C08987=1026.109,2.231,-95.350,167.487,46.558,158.592
C08988=1026.114,2.480,-95.365,167.491,46.555,158.592
C08989=1026.122,2.729,-95.379,167.493,46.552,158.592
C08990=1026.127,2.979,-95.393,167.495,46.549,158.592
C08991=1026.133,3.228,-95.408,167.498,46.546,158.592
C08992=1026.139,3.477,-95.423,167.501,46.544,158.592
C08993=1026.146,3.727,-95.438,167.503,46.541,158.591
C08994=1026.151,3.977,-95.452,167.506,46.538,158.591
C08995=1026.157,4.226,-95.467,167.509,46.535,158.591
C08996=1026.164,4.476,-95.481,167.511,46.533,158.591
C08997=1026.170,4.725,-95.496,167.514,46.530,158.590
C08998=1026.176,4.975,-95.510,167.516,46.527,158.590
C08999=1026.181,5.224,-95.525,167.519,46.524,158.590
C09000=1026.188,5.474,-95.540,167.522,46.521,158.590
C09001=1026.194,5.723,-95.555,167.524,46.519,158.590
C09002=1026.200,5.973,-95.568,167.527,46.516,158.589
C09003=1026.207,6.222,-95.583,167.530,46.513,158.589
C09004=1026.213,6.471,-95.598,167.532,46.510,158.589
C09005=1026.219,6.721,-95.612,167.534,46.507,158.589
C09006=1026.225,6.971,-95.627,167.538,46.504,158.589
C09007=1026.231,7.219,-95.642,167.540,46.502,158.588
C09008=1026.237,7.470,-95.656,167.542,46.499,158.588
C09009=1026.244,7.719,-95.671,167.545,46.496,158.588
C09010=1026.249,7.968,-95.686,167.548,46.493,158.588
C09011=1026.256,8.218,-95.701,167.550,46.490,158.587
C09012=1026.262,8.468,-95.716,167.553,46.487,158.587
C09013=1026.268,8.717,-95.730,167.555,46.485,158.587
C09014=1026.274,8.967,-95.744,167.559,46.482,158.587
C09015=1026.280,9.217,-95.759,167.561,46.479,158.587
C09016=1026.286,9.466,-95.774,167.563,46.477,158.586
C09017=1026.293,9.715,-95.789,167.567,46.474,158.586
C09018=1026.299,9.965,-95.804,167.569,46.471,158.586
C09019=1026.306,10.214,-95.818,167.571,46.468,158.586
C09020=1026.312,10.463,-95.833,167.574,46.465,158.586
C09021=1026.318,10.713,-95.848,167.577,46.462,158.585
C09022=1026.325,10.962,-95.863,167.579,46.459,158.585
C09023=1026.331,11.246,-95.880,167.582,46.456,158.585
C09024=1026.339,11.530,-95.896,167.585,46.453,158.585
C09025=1026.346,11.815,-95.914,167.588,46.450,158.584
C09026=1026.353,12.098,-95.930,167.591,46.446,158.584
C09027=1026.359,12.348,-95.945,167.594,46.443,158.584
C09028=1026.365,12.598,-95.960,167.596,46.440,158.584
C09029=1026.371,12.847,-95.974,167.599,46.437,158.583
C09030=1026.377,13.097,-95.989,167.601,46.435,158.583
C09031=1026.384,13.347,-96.004,167.604,46.432,158.583
C09032=1026.390,13.596,-96.019,167.607,46.429,158.583
C09033=1026.396,13.845,-96.034,167.609,46.426,158.583
C09034=1026.402,14.094,-96.049,167.611,46.423,158.582
C09035=1026.408,14.344,-96.064,167.614,46.421,158.582
C09036=1026.415,14.594,-96.079,167.617,46.418,158.582
C09037=1026.420,14.843,-96.094,167.619,46.415,158.582
C09038=1026.427,15.093,-96.109,167.622,46.413,158.581
C09039=1026.432,15.343,-96.124,167.625,46.410,158.581
C09040=1026.439,15.592,-96.139,167.627,46.407,158.581
C09041=1026.445,15.841,-96.155,167.629,46.404,158.581
C09042=1026.451,16.090,-96.170,167.632,46.401,158.581
C09043=1026.458,16.340,-96.185,167.635,46.399,158.581
C09044=1026.463,16.590,-96.200,167.637,46.396,158.580
C09045=1026.470,16.839,-96.215,167.640,46.394,158.580
C09046=1026.475,17.088,-96.230,167.643,46.391,158.580
C09047=1026.482,17.337,-96.245,167.645,46.388,158.580
C09048=1026.488,17.587,-96.261,167.647,46.385,158.579
C09049=1026.494,17.837,-96.276,167.650,46.382,158.579
C09050=1026.500,18.087,-96.291,167.653,46.379,158.579
C09051=1026.507,18.335,-96.306,167.655,46.376,158.579
C09052=1026.512,18.585,-96.322,167.657,46.374,158.578
C09053=1026.519,18.835,-96.337,167.661,46.371,158.578
C09054=1026.525,19.084,-96.351,167.663,46.369,158.578
C09055=1026.532,19.333,-96.367,167.665,46.366,158.578
C09056=1026.537,19.583,-96.383,167.668,46.363,158.578
C09057=1026.543,19.832,-96.397,167.671,46.360,158.577
C09058=1026.549,20.082,-96.412,167.673,46.357,158.577
C09059=1026.555,20.331,-96.428,167.675,46.354,158.577
C09060=1026.562,20.581,-96.443,167.678,46.352,158.577
C09061=1026.567,20.831,-96.459,167.681,46.349,158.577
C09062=1026.574,21.080,-96.475,167.683,46.347,158.576
C09063=1026.581,21.330,-96.490,167.686,46.344,158.576
C09064=1026.586,21.578,-96.505,167.688,46.341,158.576
C09065=1026.592,21.828,-96.520,167.691,46.338,158.576
C09066=1026.598,22.078,-96.536,167.693,46.335,158.575
C09067=1026.605,22.327,-96.552,167.696,46.333,158.575
C09068=1026.611,22.577,-96.567,167.698,46.330,158.575
C09069=1026.617,22.827,-96.582,167.701,46.327,158.575
C09070=1026.623,23.076,-96.598,167.704,46.325,158.575
C09071=1026.629,23.326,-96.613,167.706,46.322,158.574
C09072=1026.635,23.574,-96.629,167.708,46.319,158.574
C09073=1026.641,23.824,-96.644,167.711,46.316,158.574
C09074=1026.647,24.073,-96.660,167.714,46.313,158.574
C09075=1026.654,24.323,-96.675,167.716,46.311,158.573
C09076=1026.659,24.573,-96.690,167.718,46.308,158.573
C09077=1026.666,24.822,-96.706,167.721,46.305,158.573
C09078=1026.672,25.071,-96.721,167.724,46.302,158.573
C09079=1026.678,25.321,-96.737,167.726,46.299,158.573
C09080=1026.685,25.570,-96.752,167.729,46.296,158.572
C09081=1026.691,25.820,-96.768,167.732,46.294,158.572
C09082=1026.697,26.069,-96.783,167.734,46.292,158.572
C09083=1026.703,26.319,-96.800,167.736,46.289,158.572
C09084=1026.709,26.568,-96.814,167.739,46.286,158.572
C09085=1026.716,26.817,-96.830,167.742,46.283,158.571
C09086=1026.721,27.067,-96.845,167.744,46.280,158.571
C09087=1026.729,27.352,-96.863,167.747,46.277,158.571
C09088=1026.736,27.637,-96.881,167.749,46.274,158.570
C09089=1026.742,27.923,-96.900,167.752,46.271,158.570
C09090=1026.750,28.208,-96.917,167.756,46.268,158.570
C09091=1026.756,28.458,-96.933,167.758,46.265,158.570
C09092=1026.761,28.707,-96.949,167.760,46.262,158.570
C09093=1026.768,28.956,-96.965,167.762,46.260,158.569
C09094=1026.774,29.206,-96.980,167.766,46.257,158.569
C09095=1026.780,29.455,-96.996,167.768,46.254,158.569
C09096=1026.786,29.705,-97.012,167.770,46.252,158.569
C09097=1026.792,29.955,-97.028,167.773,46.249,158.569
C09098=1026.799,30.204,-97.043,167.776,46.246,158.568
C09099=1026.805,30.453,-97.060,167.778,46.243,158.568
C09100=1026.810,30.703,-97.075,167.780,46.240,158.568
C09101=1026.817,30.952,-97.091,167.783,46.238,158.568
C09102=1026.823,31.201,-97.107,167.785,46.236,158.567
C09103=1026.829,31.451,-97.123,167.788,46.233,158.567
C09104=1026.835,31.700,-97.138,167.791,46.230,158.567
C09105=1026.841,31.950,-97.155,167.793,46.227,158.567
C09106=1026.847,32.199,-97.171,167.795,46.224,158.567
C09107=1026.854,32.449,-97.186,167.798,46.221,158.566
C09108=1026.860,32.698,-97.202,167.801,46.219,158.566
C09109=1026.866,32.948,-97.218,167.803,46.216,158.566
C09110=1026.872,33.197,-97.234,167.805,46.213,158.566
C09111=1026.878,33.447,-97.249,167.808,46.211,158.565
C09112=1026.884,33.696,-97.266,167.811,46.208,158.565
C09113=1026.891,33.945,-97.281,167.813,46.205,158.565
C09114=1026.896,34.194,-97.298,167.815,46.203,158.565
C09115=1026.904,34.444,-97.314,167.818,46.200,158.565
C09116=1026.909,34.694,-97.329,167.821,46.197,158.564
C09117=1026.915,34.943,-97.345,167.823,46.194,158.564
C09118=1026.922,35.192,-97.361,167.825,46.191,158.564
C09119=1026.928,35.442,-97.377,167.828,46.189,158.564
C09120=1026.934,35.691,-97.394,167.830,46.186,158.563
C09121=1026.941,35.940,-97.409,167.833,46.183,158.563
C09122=1026.946,36.190,-97.425,167.836,46.180,158.563
C09123=1026.952,36.439,-97.441,167.838,46.177,158.563
C09124=1026.958,36.689,-97.457,167.840,46.175,158.562
C09125=1026.965,36.938,-97.473,167.843,46.172,158.562
C09126=1026.971,37.188,-97.490,167.846,46.170,158.562
C09127=1026.977,37.437,-97.506,167.848,46.167,158.562
C09128=1026.983,37.687,-97.522,167.850,46.164,158.562
C09129=1026.989,37.936,-97.538,167.853,46.161,158.561
C09130=1026.995,38.185,-97.555,167.856,46.158,158.561
C09131=1027.001,38.435,-97.571,167.858,46.156,158.561
C09132=1027.008,38.684,-97.587,167.861,46.153,158.561
C09133=1027.014,38.933,-97.603,167.863,46.151,158.560
C09134=1027.020,39.182,-97.619,167.865,46.148,158.560
C09135=1027.026,39.432,-97.635,167.867,46.145,158.560
C09136=1027.032,39.682,-97.652,167.871,46.142,158.560
C09137=1027.038,39.931,-97.668,167.873,46.140,158.560
C09138=1027.044,40.180,-97.684,167.875,46.137,158.559
C09139=1027.050,40.430,-97.701,167.878,46.135,158.559
C09140=1027.056,40.679,-97.717,167.880,46.132,158.559
C09141=1027.062,40.928,-97.733,167.883,46.129,158.559
C09142=1027.068,41.178,-97.749,167.885,46.126,158.558
C09143=1027.075,41.428,-97.766,167.888,46.123,158.558
C09144=1027.081,41.677,-97.782,167.890,46.121,158.558
C09145=1027.087,41.926,-97.798,167.892,46.119,158.558
C09146=1027.093,42.176,-97.814,167.895,46.116,158.558
C09147=1027.099,42.425,-97.831,167.898,46.113,158.557
C09148=1027.105,42.674,-97.847,167.900,46.110,158.557
C09149=1027.112,42.924,-97.864,167.902,46.107,158.557
C09150=1027.118,43.173,-97.880,167.905,46.105,158.557
C09151=1027.124,43.459,-97.899,167.908,46.102,158.556
C09152=1027.131,43.744,-97.918,167.910,46.099,158.556
C09153=1027.138,44.029,-97.937,167.914,46.096,158.556
C09154=1027.145,44.315,-97.956,167.916,46.093,158.556
C09155=1027.151,44.565,-97.973,167.919,46.090,158.556
C09156=1027.157,44.813,-97.990,167.921,46.088,158.555
C09157=1027.163,45.063,-98.006,167.924,46.085,158.555
C09158=1027.169,45.312,-98.022,167.926,46.083,158.555
C09159=1027.175,45.562,-98.039,167.928,46.080,158.555
C09160=1027.181,45.811,-98.056,167.931,46.077,158.554
C09161=1027.187,46.060,-98.073,167.933,46.075,158.554
C09162=1027.193,46.310,-98.089,167.936,46.072,158.554
C09163=1027.199,46.559,-98.105,167.939,46.070,158.554
C09164=1027.205,46.809,-98.123,167.941,46.067,158.554
C09165=1027.211,47.058,-98.139,167.943,46.064,158.553
C09166=1027.217,47.308,-98.156,167.946,46.062,158.553
C09167=1027.223,47.556,-98.173,167.948,46.059,158.553
C09168=1027.230,47.806,-98.189,167.950,46.057,158.553
C09169=1027.235,48.056,-98.206,167.953,46.054,158.552
C09170=1027.241,48.305,-98.223,167.956,46.051,158.552
C09171=1027.247,48.554,-98.239,167.958,46.048,158.552
C09172=1027.253,48.803,-98.256,167.961,46.046,158.552
C09173=1027.260,49.053,-98.273,167.963,46.043,158.552
C09174=1027.265,49.303,-98.290,167.965,46.041,158.551
C09175=1027.271,49.552,-98.306,167.967,46.038,158.551
C09176=1027.277,49.801,-98.323,167.971,46.035,158.551
C09177=1027.284,50.051,-98.340,167.973,46.033,158.551
C09178=1027.290,50.299,-98.357,167.975,46.030,158.550
C09179=1027.295,50.549,-98.373,167.978,46.027,158.550
C09180=1027.302,50.799,-98.390,167.980,46.025,158.550
C09181=1027.308,51.048,-98.407,167.982,46.022,158.550
C09182=1027.314,51.297,-98.423,167.984,46.019,158.549
C09183=1027.320,51.546,-98.440,167.988,46.016,158.549
C09184=1027.326,51.796,-98.457,167.990,46.014,158.549
C09185=1027.332,52.045,-98.474,167.992,46.011,158.549
C09186=1027.338,52.294,-98.491,167.995,46.009,158.549
C09187=1027.345,52.544,-98.507,167.997,46.006,158.548
C09188=1027.350,52.793,-98.525,167.999,46.003,158.548
C09189=1027.356,53.043,-98.541,168.002,46.000,158.548
C09190=1027.363,53.292,-98.558,168.005,45.997,158.548
C09191=1027.369,53.542,-98.575,168.007,45.995,158.547
C09192=1027.375,53.790,-98.592,168.009,45.993,158.547
C09193=1027.381,54.041,-98.609,168.012,45.990,158.547
C09194=1027.387,54.289,-98.626,168.014,45.987,158.547
C09195=1027.393,54.539,-98.642,168.017,45.984,158.547
C09196=1027.400,54.788,-98.659,168.020,45.982,158.546
C09197=1027.406,55.038,-98.676,168.022,45.979,158.546
C09198=1027.412,55.287,-98.693,168.024,45.976,158.546
C09199=1027.418,55.537,-98.710,168.026,45.973,158.545
C09200=1027.425,55.785,-98.727,168.030,45.970,158.545
C09201=1027.431,56.035,-98.745,168.032,45.968,158.545
C09202=1027.437,56.284,-98.761,168.034,45.965,158.545
C09203=1027.443,56.533,-98.778,168.036,45.962,158.544
C09204=1027.449,56.783,-98.795,168.039,45.960,158.544
C09205=1027.456,57.032,-98.812,168.041,45.957,158.544
C09206=1027.462,57.282,-98.829,168.044,45.954,158.544
C09207=1027.468,57.531,-98.846,168.047,45.952,158.544
C09208=1027.474,57.780,-98.863,168.049,45.949,158.543
C09209=1027.481,58.030,-98.879,168.051,45.946,158.543
C09210=1027.486,58.279,-98.897,168.053,45.944,158.543
C09211=1027.493,58.529,-98.914,168.057,45.941,158.543
C09212=1027.499,58.778,-98.931,168.059,45.938,158.542
C09213=1027.505,59.026,-98.948,168.061,45.935,158.542
C09214=1027.511,59.277,-98.965,168.064,45.932,158.542
C09215=1027.518,59.562,-98.984,168.067,45.929,158.542
C09216=1027.526,59.847,-99.004,168.069,45.926,158.541
C09217=1027.532,60.132,-99.023,168.072,45.923,158.541
C09218=1027.540,60.417,-99.042,168.075,45.919,158.541
C09219=1027.546,60.666,-99.060,168.077,45.917,158.540
C09220=1027.552,60.916,-99.077,168.080,45.914,158.540
C09221=1027.559,61.165,-99.094,168.082,45.911,158.540
C09222=1027.565,61.414,-99.111,168.085,45.908,158.540
C09223=1027.571,61.664,-99.128,168.087,45.906,158.539
C09224=1027.577,61.913,-99.145,168.090,45.903,158.539
C09225=1027.584,62.163,-99.162,168.092,45.900,158.539
C09226=1027.590,62.411,-99.179,168.094,45.897,158.539
C09227=1027.597,62.661,-99.196,168.097,45.894,158.538
C09228=1027.602,62.910,-99.214,168.100,45.892,158.538
C09229=1027.609,63.160,-99.231,168.102,45.889,158.538
C09230=1027.615,63.409,-99.247,168.104,45.886,158.538
C09231=1027.621,63.659,-99.265,168.107,45.884,158.537
C09232=1027.627,63.908,-99.282,168.110,45.881,158.537
C09233=1027.633,64.157,-99.300,168.112,45.879,158.537
C09234=1027.640,64.406,-99.317,168.115,45.876,158.537
C09235=1027.646,64.656,-99.335,168.117,45.873,158.537
C09236=1027.652,64.905,-99.352,168.119,45.870,158.536
C09237=1027.658,65.154,-99.370,168.121,45.868,158.536
C09238=1027.663,65.404,-99.387,168.125,45.865,158.536
C09239=1027.670,65.653,-99.404,168.127,45.862,158.536
C09240=1027.676,65.902,-99.422,168.129,45.859,158.535
C09241=1027.683,66.152,-99.439,168.132,45.857,158.535
C09242=1027.688,66.401,-99.457,168.134,45.855,158.535
C09243=1027.695,66.650,-99.474,168.136,45.852,158.535
C09244=1027.700,66.899,-99.491,168.139,45.849,158.534
C09245=1027.707,67.149,-99.509,168.142,45.846,158.534
C09246=1027.713,67.398,-99.526,168.144,45.843,158.534
C09247=1027.719,67.648,-99.544,168.146,45.841,158.534
C09248=1027.725,67.896,-99.561,168.149,45.838,158.533
C09249=1027.731,68.146,-99.579,168.151,45.835,158.533
C09250=1027.737,68.396,-99.597,168.153,45.833,158.533
C09251=1027.744,68.644,-99.614,168.157,45.830,158.533
C09252=1027.750,68.894,-99.632,168.159,45.828,158.533
C09253=1027.755,69.143,-99.650,168.161,45.825,158.532
C09254=1027.762,69.393,-99.667,168.163,45.822,158.532
C09255=1027.768,69.642,-99.684,168.166,45.819,158.532
C09256=1027.774,69.891,-99.702,168.168,45.817,158.532
C09257=1027.779,70.141,-99.720,168.171,45.815,158.531
C09258=1027.786,70.390,-99.737,168.173,45.812,158.531
C09259=1027.792,70.640,-99.755,168.176,45.809,158.531
C09260=1027.798,70.889,-99.773,168.178,45.806,158.531
C09261=1027.804,71.138,-99.791,168.181,45.804,158.530
C09262=1027.811,71.387,-99.808,168.183,45.801,158.530
C09263=1027.817,71.636,-99.826,168.185,45.799,158.530
C09264=1027.822,71.885,-99.844,168.188,45.796,158.530
C09265=1027.828,72.135,-99.862,168.190,45.793,158.529
C09266=1027.835,72.385,-99.879,168.193,45.791,158.529
C09267=1027.841,72.634,-99.897,168.195,45.788,158.529
C09268=1027.847,72.883,-99.915,168.198,45.785,158.529
C09269=1027.853,73.132,-99.933,168.200,45.783,158.529
C09270=1027.859,73.381,-99.951,168.203,45.780,158.528
C09271=1027.866,73.631,-99.968,168.205,45.778,158.528
C09272=1027.871,73.880,-99.986,168.207,45.775,158.528
C09273=1027.877,74.130,-100.004,168.210,45.772,158.528
C09274=1027.883,74.378,-100.022,168.213,45.769,158.527
C09275=1027.889,74.628,-100.040,168.215,45.767,158.527
C09276=1027.896,74.877,-100.057,168.217,45.764,158.527
C09277=1027.902,75.126,-100.075,168.220,45.762,158.527
C09278=1027.908,75.376,-100.093,168.222,45.759,158.526
C09279=1027.915,75.661,-100.113,168.225,45.756,158.526
C09280=1027.922,75.946,-100.134,168.228,45.753,158.526
C09281=1027.929,76.231,-100.154,168.231,45.750,158.526
C09282=1027.936,76.516,-100.175,168.234,45.746,158.525
C09283=1027.942,76.766,-100.193,168.236,45.744,158.525
C09284=1027.948,77.015,-100.211,168.238,45.742,158.525
C09285=1027.954,77.264,-100.229,168.241,45.739,158.525
C09286=1027.960,77.513,-100.246,168.243,45.736,158.524
C09287=1027.967,77.762,-100.265,168.246,45.733,158.524
C09288=1027.972,78.011,-100.282,168.248,45.730,158.524
C09289=1027.979,78.261,-100.300,168.251,45.728,158.524
C09290=1027.984,78.511,-100.320,168.253,45.726,158.523
C09291=1027.990,78.760,-100.337,168.256,45.723,158.523
C09292=1027.996,79.009,-100.356,168.258,45.720,158.523
C09293=1028.002,79.258,-100.374,168.260,45.718,158.523
C09294=1028.008,79.507,-100.392,168.263,45.716,158.522
C09295=1028.014,79.757,-100.410,168.265,45.713,158.522
C09296=1028.020,80.006,-100.428,168.268,45.710,158.522
C09297=1028.026,80.255,-100.446,168.270,45.707,158.522
C09298=1028.032,80.505,-100.464,168.273,45.705,158.522
C09299=1028.039,80.754,-100.483,168.275,45.703,158.521
C09300=1028.044,81.003,-100.500,168.278,45.700,158.521
C09301=1028.051,81.252,-100.519,168.280,45.697,158.521
C09302=1028.057,81.502,-100.537,168.282,45.694,158.520
C09303=1028.063,81.751,-100.556,168.285,45.692,158.520
C09304=1028.068,82.000,-100.574,168.288,45.689,158.520
C09305=1028.074,82.249,-100.592,168.290,45.687,158.520
C09306=1028.081,82.499,-100.610,168.292,45.684,158.520
C09307=1028.086,82.747,-100.629,168.295,45.681,158.519
C09308=1028.092,82.997,-100.647,168.297,45.679,158.519
C09309=1028.099,83.246,-100.665,168.299,45.677,158.519
C09310=1028.105,83.496,-100.683,168.302,45.674,158.519
C09311=1028.111,83.744,-100.701,168.305,45.671,158.518
C09312=1028.117,83.994,-100.719,168.307,45.668,158.518
C09313=1028.123,84.243,-100.738,168.310,45.666,158.518
C09314=1028.130,84.492,-100.757,168.312,45.663,158.518
C09315=1028.135,84.741,-100.774,168.314,45.661,158.518
C09316=1028.141,84.991,-100.793,168.317,45.658,158.517
C09317=1028.147,85.241,-100.811,168.320,45.655,158.517
C09318=1028.154,85.490,-100.830,168.322,45.653,158.517
C09319=1028.160,85.739,-100.848,168.325,45.650,158.517
C09320=1028.166,85.988,-100.866,168.327,45.647,158.516
C09321=1028.172,86.237,-100.885,168.329,45.645,158.516
C09322=1028.178,86.487,-100.903,168.332,45.642,158.516
C09323=1028.184,86.736,-100.921,168.335,45.640,158.516
C09324=1028.191,86.985,-100.940,168.337,45.637,158.515
C09325=1028.196,87.234,-100.958,168.339,45.634,158.515
C09326=1028.203,87.483,-100.976,168.342,45.631,158.515
C09327=1028.209,87.732,-100.996,168.344,45.629,158.515
C09328=1028.215,87.982,-101.014,168.346,45.626,158.514
C09329=1028.221,88.231,-101.032,168.350,45.623,158.514
C09330=1028.227,88.481,-101.050,168.352,45.620,158.514
C09331=1028.233,88.730,-101.068,168.354,45.618,158.514
C09332=1028.239,88.979,-101.087,168.357,45.616,158.513
C09333=1028.246,89.228,-101.106,168.359,45.613,158.513
C09334=1028.252,89.477,-101.124,168.361,45.610,158.513
C09335=1028.258,89.727,-101.143,168.364,45.607,158.513
C09336=1028.264,89.976,-101.162,168.367,45.605,158.512
C09337=1028.271,90.225,-101.180,168.369,45.603,158.512
C09338=1028.275,90.475,-101.198,168.372,45.600,158.512
C09339=1028.282,90.724,-101.217,168.374,45.597,158.512
C09340=1028.287,90.973,-101.236,168.376,45.595,158.511
C09341=1028.294,91.222,-101.255,168.379,45.593,158.511
C09342=1028.300,91.471,-101.273,168.382,45.590,158.511
C09343=1028.307,91.757,-101.295,168.384,45.587,158.511
C09344=1028.313,92.041,-101.316,168.387,45.583,158.510
C09345=1028.321,92.326,-101.338,168.390,45.581,158.510
C09346=1028.327,92.612,-101.359,168.393,45.578,158.510
C09347=1028.334,92.861,-101.378,168.395,45.575,158.510
C09348=1028.339,93.110,-101.397,168.398,45.573,158.510
C09349=1028.345,93.358,-101.415,168.400,45.570,158.509
C09350=1028.351,93.608,-101.434,168.402,45.568,158.509
C09351=1028.357,93.857,-101.453,168.405,45.565,158.509
C09352=1028.364,94.106,-101.472,168.408,45.562,158.509
C09353=1028.369,94.356,-101.491,168.410,45.560,158.508
C09354=1028.376,94.605,-101.510,168.413,45.557,158.508
C09355=1028.381,94.854,-101.529,168.415,45.555,158.508
C09356=1028.388,95.104,-101.547,168.417,45.552,158.508
C09357=1028.394,95.353,-101.565,168.420,45.549,158.507
C09358=1028.399,95.602,-101.584,168.423,45.547,158.507
C09359=1028.406,95.851,-101.603,168.425,45.544,158.507
C09360=1028.411,96.100,-101.622,168.427,45.542,158.507
C09361=1028.418,96.349,-101.641,168.430,45.539,158.506
C09362=1028.424,96.599,-101.660,168.432,45.536,158.506
C09363=1028.430,96.848,-101.679,168.435,45.534,158.506
C09364=1028.436,97.097,-101.697,168.438,45.532,158.506
C09365=1028.442,97.347,-101.717,168.440,45.529,158.506
C09366=1028.448,97.596,-101.735,168.442,45.526,158.505
C09367=1028.454,97.845,-101.755,168.445,45.523,158.505
C09368=1028.460,98.094,-101.773,168.448,45.521,158.505
C09369=1028.467,98.343,-101.792,168.450,45.518,158.505
C09370=1028.473,98.593,-101.811,168.453,45.516,158.504
C09371=1028.479,98.842,-101.830,168.455,45.513,158.504
C09372=1028.485,99.091,-101.850,168.457,45.510,158.504
C09373=1028.491,99.340,-101.868,168.460,45.508,158.504
C09374=1028.498,99.589,-101.887,168.463,45.505,158.503
C09375=1028.503,99.838,-101.906,168.465,45.502,158.503
C09376=1028.509,100.088,-101.925,168.468,45.500,158.503
C09377=1028.516,100.337,-101.944,168.470,45.498,158.503
C09378=1028.521,100.586,-101.963,168.472,45.495,158.502
C09379=1028.527,100.836,-101.983,168.475,45.492,158.502
C09380=1028.534,101.084,-102.002,168.478,45.490,158.502
C09381=1028.539,101.334,-102.021,168.480,45.487,158.502
C09382=1028.545,101.583,-102.040,168.483,45.485,158.502
C09383=1028.551,101.833,-102.060,168.485,45.483,158.501
C09384=1028.557,102.082,-102.078,168.488,45.480,158.501
C09385=1028.563,102.331,-102.098,168.490,45.477,158.501
C09386=1028.569,102.580,-102.118,168.492,45.475,158.501
C09387=1028.575,102.829,-102.136,168.496,45.472,158.501
C09388=1028.581,103.079,-102.155,168.498,45.470,158.500
C09389=1028.587,103.327,-102.175,168.500,45.467,158.500
C09390=1028.593,103.576,-102.194,168.503,45.465,158.500
C09391=1028.599,103.826,-102.213,168.505,45.462,158.500
C09392=1028.605,104.075,-102.233,168.507,45.460,158.499
C09393=1028.611,104.324,-102.252,168.511,45.457,158.499
C09394=1028.617,104.573,-102.271,168.513,45.455,158.499
C09395=1028.623,104.823,-102.290,168.515,45.452,158.499
C09396=1028.629,105.071,-102.310,168.518,45.449,158.498
C09397=1028.635,105.321,-102.329,168.520,45.447,158.498
C09398=1028.641,105.570,-102.348,168.523,45.444,158.498
C09399=1028.647,105.819,-102.368,168.526,45.442,158.498
C09400=1028.653,106.068,-102.387,168.528,45.439,158.498
C09401=1028.659,106.317,-102.406,168.530,45.436,158.497
C09402=1028.665,106.566,-102.426,168.533,45.434,158.497
C09403=1028.671,106.816,-102.445,168.535,45.432,158.497
C09404=1028.678,107.064,-102.465,168.539,45.429,158.497
C09405=1028.683,107.314,-102.484,168.541,45.426,158.496
C09406=1028.689,107.563,-102.503,168.543,45.423,158.496
C09407=1028.696,107.849,-102.525,168.546,45.421,158.496
C09408=1028.703,108.133,-102.548,168.549,45.418,158.496
C09409=1028.710,108.418,-102.570,168.552,45.415,158.495
C09410=1028.717,108.703,-102.592,168.555,45.412,158.495
C09411=1028.723,108.952,-102.612,168.558,45.409,158.495
C09412=1028.729,109.201,-102.631,168.560,45.407,158.495
C09413=1028.735,109.450,-102.650,168.562,45.404,158.494
C09414=1028.741,109.699,-102.670,168.565,45.401,158.494
C09415=1028.748,109.949,-102.690,168.568,45.399,158.494
C09416=1028.754,110.198,-102.710,168.570,45.397,158.494
C09417=1028.760,110.447,-102.728,168.573,45.394,158.493
C09418=1028.766,110.696,-102.748,168.575,45.391,158.493
C09419=1028.772,110.946,-102.767,168.578,45.389,158.493
C09420=1028.778,111.194,-102.787,168.581,45.386,158.493
C09421=1028.783,111.444,-102.807,168.583,45.384,158.492
C09422=1028.789,111.693,-102.827,168.585,45.381,158.492
C09423=1028.796,111.942,-102.847,168.588,45.379,158.492
C09424=1028.802,112.192,-102.866,168.591,45.376,158.492
C09425=1028.808,112.440,-102.886,168.593,45.373,158.492
C09426=1028.813,112.690,-102.905,168.596,45.371,158.491
C09427=1028.820,112.938,-102.925,168.598,45.369,158.491
C09428=1028.825,113.188,-102.945,168.600,45.366,158.491
C09429=1028.832,113.438,-102.965,168.604,45.364,158.491
C09430=1028.838,113.686,-102.985,168.606,45.361,158.491
C09431=1028.844,113.935,-103.005,168.609,45.359,158.490
C09432=1028.849,114.185,-103.024,168.611,45.357,158.490
C09433=1028.855,114.434,-103.045,168.613,45.354,158.490
C09434=1028.860,114.683,-103.064,168.616,45.352,158.490
C09435=1028.866,114.932,-103.084,168.619,45.349,158.490
C09436=1028.873,115.182,-103.104,168.622,45.346,158.489
C09437=1028.879,115.430,-103.124,168.624,45.344,158.489
C09438=1028.885,115.679,-103.144,168.626,45.342,158.489
C09439=1028.890,115.929,-103.164,168.629,45.340,158.489
C09440=1028.896,116.178,-103.184,168.631,45.337,158.488
C09441=1028.902,116.427,-103.204,168.635,45.334,158.488
C09442=1028.908,116.676,-103.224,168.637,45.332,158.488
C09443=1028.914,116.925,-103.244,168.639,45.329,158.488
C09444=1028.919,117.175,-103.264,168.642,45.327,158.488
C09445=1028.925,117.423,-103.284,168.644,45.325,158.487
C09446=1028.931,117.672,-103.304,168.647,45.322,158.487
C09447=1028.938,117.922,-103.324,168.650,45.320,158.487
C09448=1028.944,118.171,-103.344,168.652,45.317,158.487
C09449=1028.949,118.420,-103.365,168.655,45.315,158.486
C09450=1028.955,118.669,-103.384,168.657,45.313,158.486
C09451=1028.961,118.918,-103.404,168.660,45.310,158.486
C09452=1028.967,119.167,-103.424,168.663,45.308,158.486
C09453=1028.973,119.416,-103.444,168.665,45.305,158.486
C09454=1028.979,119.665,-103.465,168.668,45.302,158.485
C09455=1028.985,119.914,-103.485,168.670,45.300,158.485
C09456=1028.991,120.164,-103.505,168.673,45.298,158.485
C09457=1028.997,120.413,-103.524,168.676,45.295,158.485
C09458=1029.003,120.662,-103.544,168.678,45.293,158.485
C09459=1029.008,120.911,-103.565,168.681,45.290,158.484
C09460=1029.015,121.161,-103.585,168.684,45.287,158.484
C09461=1029.021,121.409,-103.605,168.686,45.285,158.484
C09462=1029.027,121.658,-103.625,168.689,45.283,158.484
C09463=1029.033,121.907,-103.645,168.691,45.280,158.483
C09464=1029.039,122.157,-103.666,168.695,45.278,158.483
C09465=1029.045,122.406,-103.686,168.697,45.275,158.483
C09466=1029.051,122.654,-103.706,168.699,45.272,158.483
C09467=1029.057,122.904,-103.726,168.702,45.270,158.483
C09468=1029.063,123.153,-103.746,168.705,45.268,158.482
C09469=1029.068,123.402,-103.767,168.707,45.265,158.482
C09470=1029.075,123.651,-103.787,168.710,45.263,158.482
C09471=1029.082,123.936,-103.810,168.713,45.260,158.482
C09472=1029.089,124.220,-103.833,168.715,45.257,158.482
C09473=1029.096,124.506,-103.857,168.719,45.255,158.481
C09474=1029.103,124.790,-103.879,168.722,45.251,158.481
C09475=1029.109,125.039,-103.899,168.724,45.249,158.481
C09476=1029.115,125.289,-103.920,168.727,45.246,158.481
C09477=1029.121,125.538,-103.940,168.730,45.244,158.480
C09478=1029.127,125.787,-103.960,168.732,45.242,158.480
C09479=1029.133,126.036,-103.980,168.735,45.239,158.480
C09480=1029.139,126.285,-104.000,168.738,45.236,158.480
C09481=1029.144,126.534,-104.021,168.741,45.234,158.480
C09482=1029.151,126.783,-104.041,168.743,45.231,158.479
C09483=1029.157,127.032,-104.061,168.745,45.229,158.479
C09484=1029.164,127.282,-104.081,168.749,45.226,158.479
C09485=1029.169,127.531,-104.102,168.751,45.224,158.479
C09486=1029.175,127.780,-104.122,168.753,45.221,158.478
C09487=1029.181,128.029,-104.142,168.757,45.218,158.478
C09488=1029.188,128.277,-104.163,168.759,45.216,158.478
C09489=1029.194,128.527,-104.184,168.761,45.214,158.478
C09490=1029.200,128.776,-104.204,168.765,45.211,158.477
C09491=1029.206,129.025,-104.224,168.767,45.209,158.477
C09492=1029.212,129.274,-104.244,168.770,45.206,158.477
C09493=1029.217,129.524,-104.265,168.773,45.203,158.477
C09494=1029.224,129.773,-104.285,168.775,45.201,158.477
C09495=1029.230,130.021,-104.306,168.778,45.199,158.476
C09496=1029.237,130.271,-104.326,168.781,45.196,158.476
C09497=1029.242,130.520,-104.347,168.783,45.193,158.476
C09498=1029.248,130.769,-104.367,168.786,45.191,158.476
C09499=1029.254,131.018,-104.388,168.788,45.189,158.476
C09500=1029.260,131.267,-104.408,168.792,45.186,158.475
C09501=1029.266,131.517,-104.429,168.794,45.184,158.475
C09502=1029.272,131.765,-104.450,168.797,45.182,158.475
C09503=1029.278,132.015,-104.471,168.799,45.179,158.475
C09504=1029.284,132.263,-104.491,168.802,45.176,158.475
C09505=1029.290,132.512,-104.512,168.805,45.174,158.474
C09506=1029.296,132.762,-104.533,168.807,45.172,158.474
C09507=1029.302,133.005,-104.552,168.811,45.169,158.474
C09508=1029.308,133.250,-104.573,168.813,45.167,158.474
C09509=1029.314,133.493,-104.594,168.815,45.165,158.474
C09510=1029.319,133.737,-104.614,168.818,45.162,158.473
C09511=1029.325,133.982,-104.634,168.820,45.160,158.473
C09512=1029.331,134.226,-104.655,168.824,45.157,158.473
C09513=1029.337,134.469,-104.675,168.826,45.155,158.473
C09514=1029.343,134.713,-104.695,168.828,45.153,158.473
C09515=1029.348,134.963,-104.716,168.831,45.151,158.472
C09516=1029.355,135.212,-104.737,168.834,45.148,158.472
C09517=1029.360,135.461,-104.757,168.837,45.146,158.472
C09518=1029.367,135.710,-104.778,168.839,45.143,158.472
C09519=1029.372,135.959,-104.799,168.842,45.140,158.472
C09520=1029.379,136.208,-104.821,168.845,45.138,158.471
C09521=1029.385,136.457,-104.841,168.847,45.136,158.471
C09522=1029.391,136.706,-104.862,168.851,45.133,158.471
C09523=1029.397,136.956,-104.883,168.853,45.131,158.471
C09524=1029.403,137.204,-104.904,168.856,45.129,158.471
C09525=1029.409,137.454,-104.925,168.859,45.126,158.470
C09526=1029.414,137.702,-104.946,168.862,45.124,158.470
C09527=1029.421,137.952,-104.966,168.864,45.121,158.470
C09528=1029.427,138.200,-104.988,168.867,45.119,158.470
C09529=1029.432,138.450,-105.008,168.870,45.117,158.470
C09530=1029.439,138.698,-105.029,168.872,45.115,158.469
C09531=1029.445,138.947,-105.051,168.876,45.112,158.469
C09532=1029.450,139.197,-105.071,168.878,45.110,158.469
C09533=1029.456,139.446,-105.093,168.880,45.107,158.469
C09534=1029.462,139.695,-105.114,168.883,45.105,158.469
C09535=1029.470,139.989,-105.139,168.886,45.102,158.468
C09536=1029.477,140.284,-105.164,168.890,45.099,158.468
C09537=1029.483,140.579,-105.189,168.893,45.097,158.468
C09538=1029.490,140.874,-105.214,168.896,45.094,158.468
C09539=1029.497,141.123,-105.235,168.900,45.092,158.468
C09540=1029.502,141.372,-105.256,168.902,45.089,158.467
C09541=1029.508,141.621,-105.277,168.905,45.087,158.467
C09542=1029.514,141.870,-105.299,168.908,45.084,158.467
C09543=1029.520,142.119,-105.320,168.910,45.082,158.467
C09544=1029.525,142.368,-105.341,168.913,45.079,158.467
C09545=1029.532,142.617,-105.362,168.916,45.077,158.467
C09546=1029.538,142.866,-105.383,168.919,45.075,158.466
C09547=1029.544,143.114,-105.405,168.921,45.073,158.466
C09548=1029.550,143.364,-105.426,168.924,45.070,158.466
C09549=1029.555,143.613,-105.447,168.927,45.068,158.466
C09550=1029.562,143.862,-105.469,168.929,45.065,158.465
C09551=1029.568,144.111,-105.490,168.933,45.063,158.465
C09552=1029.574,144.360,-105.510,168.935,45.060,158.465
C09553=1029.580,144.609,-105.532,168.938,45.058,158.465
C09554=1029.586,144.858,-105.553,168.941,45.056,158.465
C09555=1029.592,145.107,-105.575,168.944,45.054,158.465
C09556=1029.598,145.356,-105.596,168.947,45.051,158.465
C09557=1029.604,145.605,-105.618,168.949,45.049,158.464
C09558=1029.610,145.854,-105.638,168.952,45.047,158.464
C09559=1029.616,146.103,-105.660,168.955,45.044,158.464
C09560=1029.622,146.353,-105.681,168.958,45.042,158.464
C09561=1029.628,146.601,-105.702,168.960,45.039,158.463
C09562=1029.634,146.850,-105.724,168.964,45.037,158.463
C09563=1029.640,147.099,-105.746,168.966,45.035,158.463
C09564=1029.646,147.348,-105.767,168.970,45.032,158.463
C09565=1029.652,147.597,-105.789,168.972,45.030,158.463
C09566=1029.658,147.846,-105.810,168.974,45.028,158.463
C09567=1029.664,148.095,-105.832,168.978,45.026,158.463
C09568=1029.670,148.344,-105.853,168.981,45.024,158.462
C09569=1029.676,148.593,-105.875,168.983,45.021,158.462
C09570=1029.681,148.842,-105.897,168.986,45.019,158.462
C09571=1029.687,149.091,-105.918,168.989,45.016,158.462
C09572=1029.693,149.341,-105.940,168.992,45.014,158.462
C09573=1029.699,149.589,-105.961,168.995,45.012,158.462
C09574=1029.705,149.838,-105.983,168.997,45.009,158.461
C09575=1029.711,150.087,-106.005,169.001,45.007,158.461
C09576=1029.717,150.337,-106.026,169.003,45.005,158.461
C09577=1029.723,150.585,-106.047,169.007,45.002,158.461
C09578=1029.729,150.834,-106.069,169.009,45.000,158.461
C09579=1029.735,151.084,-106.091,169.012,44.998,158.460
C09580=1029.740,151.332,-106.113,169.015,44.996,158.460
C09581=1029.746,151.581,-106.135,169.018,44.994,158.460
C09582=1029.752,151.830,-106.157,169.021,44.991,158.460
C09583=1029.759,152.079,-106.178,169.023,44.989,158.460
C09584=1029.764,152.328,-106.199,169.026,44.987,158.460
C09585=1029.770,152.577,-106.221,169.029,44.984,158.459
C09586=1029.776,152.826,-106.243,169.032,44.982,158.459
C09587=1029.783,153.075,-106.265,169.035,44.980,158.459
C09588=1029.788,153.324,-106.287,169.038,44.977,158.459
C09589=1029.794,153.573,-106.309,169.040,44.975,158.459
C09590=1029.800,153.822,-106.330,169.044,44.973,158.459
C09591=1029.806,154.071,-106.352,169.046,44.971,158.458
C09592=1029.813,154.320,-106.374,169.050,44.968,158.458
C09593=1029.818,154.569,-106.396,169.052,44.966,158.458
C09594=1029.824,154.818,-106.418,169.056,44.964,158.458
C09595=1029.830,155.066,-106.440,169.058,44.962,158.458
C09596=1029.836,155.316,-106.462,169.061,44.960,158.458
C09597=1029.842,155.565,-106.484,169.064,44.957,158.458
C09598=1029.847,155.814,-106.505,169.067,44.955,158.457
C09599=1029.854,156.098,-106.531,169.070,44.953,158.457
C09600=1029.862,156.382,-106.556,169.073,44.950,158.457
C09601=1029.868,156.667,-106.581,169.077,44.947,158.457
C09602=1029.875,156.951,-106.606,169.080,44.945,158.457
C09603=1029.881,157.200,-106.628,169.083,44.943,158.456
C09604=1029.887,157.449,-106.650,169.086,44.940,158.456
C09605=1029.893,157.698,-106.672,169.089,44.938,158.456
C09606=1029.898,157.947,-106.694,169.092,44.936,158.456
C09607=1029.905,158.196,-106.716,169.095,44.933,158.456
C09608=1029.910,158.445,-106.738,169.098,44.931,158.456
C09609=1029.917,158.694,-106.761,169.101,44.929,158.456
C09610=1029.923,158.943,-106.782,169.104,44.927,158.455
C09611=1029.929,159.192,-106.804,169.107,44.924,158.455
C09612=1029.935,159.441,-106.827,169.110,44.922,158.455
C09613=1029.940,159.689,-106.848,169.113,44.920,158.455
C09614=1029.946,159.938,-106.871,169.115,44.918,158.455
C09615=1029.951,160.188,-106.893,169.119,44.916,158.455
C09616=1029.958,160.436,-106.916,169.121,44.914,158.455
C09617=1029.964,160.685,-106.939,169.125,44.912,158.454
C09618=1029.969,160.935,-106.961,169.127,44.910,158.454
C09619=1029.975,161.184,-106.984,169.130,44.907,158.454
C09620=1029.981,161.432,-107.006,169.133,44.905,158.454
C09621=1029.986,161.681,-107.028,169.136,44.903,158.454
C09622=1029.992,161.930,-107.051,169.139,44.901,158.454
C09623=1029.998,162.179,-107.073,169.142,44.899,158.454
C09624=1030.004,162.428,-107.096,169.146,44.897,158.454
C09625=1030.009,162.677,-107.118,169.148,44.895,158.453
C09626=1030.015,162.926,-107.141,169.151,44.893,158.453
C09627=1030.021,163.174,-107.163,169.154,44.891,158.453
C09628=1030.026,163.423,-107.186,169.157,44.889,158.453
C09629=1030.032,163.672,-107.209,169.160,44.887,158.453
C09630=1030.038,163.922,-107.231,169.163,44.885,158.453
C09631=1030.044,164.170,-107.253,169.167,44.883,158.453
C09632=1030.050,164.419,-107.276,169.169,44.881,158.453
C09633=1030.056,164.668,-107.299,169.173,44.878,158.452
C09634=1030.062,164.917,-107.321,169.175,44.877,158.452
C09635=1030.067,165.166,-107.344,169.179,44.874,158.452
C09636=1030.073,165.415,-107.367,169.181,44.872,158.452
C09637=1030.079,165.664,-107.390,169.184,44.870,158.452
C09638=1030.085,165.913,-107.412,169.187,44.868,158.452
C09639=1030.090,166.161,-107.434,169.190,44.866,158.452
C09640=1030.096,166.410,-107.457,169.193,44.864,158.452
C09641=1030.102,166.659,-107.480,169.196,44.862,158.451
C09642=1030.108,166.908,-107.502,169.199,44.859,158.451
C09643=1030.114,167.157,-107.525,169.202,44.857,158.451
C09644=1030.120,167.406,-107.548,169.206,44.855,158.451
C09645=1030.125,167.655,-107.570,169.208,44.853,158.451
C09646=1030.131,167.904,-107.592,169.212,44.851,158.451
C09647=1030.137,168.153,-107.615,169.214,44.849,158.451
C09648=1030.143,168.401,-107.638,169.218,44.847,158.451
C09649=1030.149,168.650,-107.661,169.220,44.845,158.450
C09650=1030.155,168.899,-107.684,169.224,44.843,158.450
C09651=1030.161,169.148,-107.707,169.227,44.841,158.450
C09652=1030.167,169.397,-107.730,169.230,44.839,158.450
C09653=1030.172,169.646,-107.752,169.234,44.837,158.450
C09654=1030.179,169.895,-107.775,169.236,44.835,158.450
C09655=1030.185,170.144,-107.798,169.240,44.833,158.450
C09656=1030.191,170.393,-107.821,169.242,44.831,158.450
C09657=1030.196,170.642,-107.843,169.246,44.828,158.450
C09658=1030.202,170.891,-107.866,169.248,44.826,158.449
C09659=1030.208,171.140,-107.889,169.252,44.824,158.449
C09660=1030.214,171.389,-107.912,169.255,44.822,158.449
C09661=1030.220,171.638,-107.934,169.258,44.820,158.449
C09662=1030.226,171.886,-107.957,169.261,44.817,158.449
C09663=1030.233,172.170,-107.984,169.265,44.815,158.449
C09664=1030.240,172.454,-108.010,169.269,44.813,158.449
C09665=1030.246,172.738,-108.036,169.272,44.810,158.448
C09666=1030.254,173.022,-108.062,169.275,44.808,158.448
C09667=1030.259,173.271,-108.085,169.278,44.806,158.448
C09668=1030.265,173.519,-108.108,169.282,44.804,158.448
C09669=1030.271,173.768,-108.130,169.285,44.802,158.448
C09670=1030.278,174.018,-108.153,169.288,44.800,158.448
C09671=1030.284,174.267,-108.176,169.291,44.798,158.448
C09672=1030.289,174.515,-108.199,169.294,44.796,158.448
C09673=1030.295,174.764,-108.223,169.297,44.794,158.448
C09674=1030.302,175.012,-108.245,169.301,44.791,158.448
C09675=1030.307,175.261,-108.268,169.304,44.790,158.447
C09676=1030.314,175.511,-108.292,169.307,44.787,158.447
C09677=1030.320,175.760,-108.315,169.311,44.785,158.447
C09678=1030.325,176.009,-108.338,169.313,44.783,158.447
C09679=1030.332,176.257,-108.360,169.317,44.781,158.447
C09680=1030.338,176.505,-108.384,169.319,44.779,158.447
C09681=1030.344,176.755,-108.407,169.323,44.777,158.447
C09682=1030.350,177.004,-108.430,169.326,44.775,158.447
C09683=1030.356,177.253,-108.453,169.329,44.773,158.447
C09684=1030.362,177.501,-108.475,169.333,44.771,158.446
C09685=1030.368,177.750,-108.499,169.336,44.769,158.446
C09686=1030.374,177.999,-108.522,169.339,44.767,158.446
C09687=1030.380,178.248,-108.545,169.342,44.765,158.446
C09688=1030.386,178.497,-108.568,169.346,44.762,158.446
C09689=1030.393,178.745,-108.591,169.348,44.760,158.446
C09690=1030.399,178.995,-108.614,169.352,44.758,158.446
C09691=1030.405,179.244,-108.637,169.356,44.756,158.446
C09692=1030.411,179.492,-108.661,169.358,44.754,158.446
C09693=1030.417,179.741,-108.684,169.362,44.752,158.445
C09694=1030.424,179.990,-108.707,169.365,44.750,158.445
C09695=1030.430,180.238,-108.730,169.368,44.748,158.445
C09696=1030.435,180.487,-108.753,169.371,44.746,158.445
C09697=1030.442,180.737,-108.777,169.375,44.744,158.445
C09698=1030.448,180.985,-108.800,169.379,44.741,158.445
C09699=1030.453,181.234,-108.823,169.381,44.740,158.445
C09700=1030.461,181.483,-108.846,169.385,44.737,158.445
C09701=1030.467,181.732,-108.870,169.388,44.735,158.445
C09702=1030.472,181.980,-108.892,169.391,44.733,158.444
C09703=1030.479,182.230,-108.916,169.394,44.731,158.444
C09704=1030.485,182.478,-108.939,169.398,44.729,158.444
C09705=1030.490,182.727,-108.962,169.401,44.727,158.444
C09706=1030.498,182.976,-108.986,169.404,44.725,158.444
C09707=1030.503,183.225,-109.009,169.408,44.723,158.444
C09708=1030.509,183.473,-109.033,169.411,44.721,158.444
C09709=1030.515,183.723,-109.058,169.414,44.719,158.444
C09710=1030.520,183.972,-109.081,169.418,44.718,158.444
C09711=1030.526,184.220,-109.105,169.420,44.716,158.444
C09712=1030.532,184.468,-109.129,169.424,44.714,158.444
C09713=1030.538,184.718,-109.152,169.428,44.712,158.444
C09714=1030.543,184.967,-109.176,169.430,44.710,158.444
C09715=1030.549,185.215,-109.200,169.434,44.709,158.444
C09716=1030.555,185.464,-109.224,169.438,44.707,158.444
C09717=1030.561,185.713,-109.247,169.440,44.705,158.443
C09718=1030.567,185.961,-109.271,169.444,44.703,158.443
C09719=1030.573,186.211,-109.296,169.448,44.701,158.443
C09720=1030.579,186.459,-109.319,169.450,44.699,158.443
C09721=1030.584,186.708,-109.343,169.454,44.698,158.443
C09722=1030.591,186.957,-109.367,169.458,44.696,158.443
C09723=1030.596,187.206,-109.391,169.460,44.694,158.443
C09724=1030.602,187.454,-109.415,169.464,44.692,158.443
C09725=1030.609,187.703,-109.439,169.467,44.690,158.443
C09726=1030.614,187.952,-109.462,169.470,44.689,158.443
C09727=1030.620,188.236,-109.490,169.475,44.686,158.443
C09728=1030.628,188.519,-109.517,169.478,44.684,158.443
C09729=1030.635,188.802,-109.545,169.482,44.682,158.443
C09730=1030.640,189.086,-109.571,169.486,44.680,158.443
C09731=1030.647,189.335,-109.595,169.489,44.678,158.443
C09732=1030.652,189.583,-109.620,169.493,44.676,158.443
C09733=1030.659,189.832,-109.644,169.497,44.675,158.443
C09734=1030.664,190.081,-109.668,169.499,44.673,158.443
C09735=1030.671,190.330,-109.692,169.503,44.671,158.443
C09736=1030.676,190.578,-109.716,169.507,44.669,158.443
C09737=1030.683,190.827,-109.740,169.510,44.667,158.442
C09738=1030.688,191.076,-109.765,169.513,44.666,158.442
C09739=1030.694,191.324,-109.788,169.517,44.664,158.442
C09740=1030.700,191.574,-109.813,169.520,44.661,158.442
C09741=1030.706,191.822,-109.837,169.524,44.660,158.442
C09742=1030.713,192.071,-109.861,169.527,44.658,158.442
C09743=1030.718,192.319,-109.885,169.530,44.657,158.442
C09744=1030.725,192.568,-109.909,169.534,44.654,158.442
C09745=1030.730,192.817,-109.933,169.538,44.653,158.442
C09746=1030.737,193.066,-109.957,169.540,44.651,158.442
C09747=1030.742,193.315,-109.981,169.544,44.649,158.442
C09748=1030.749,193.564,-110.005,169.548,44.647,158.442
C09749=1030.754,193.812,-110.030,169.551,44.645,158.442
C09750=1030.761,194.061,-110.054,169.555,44.644,158.442
C09751=1030.766,194.310,-110.078,169.558,44.642,158.442
C09752=1030.773,194.559,-110.102,169.562,44.640,158.442
C09753=1030.778,194.808,-110.127,169.565,44.638,158.442
C09754=1030.784,195.056,-110.150,169.569,44.637,158.442
C09755=1030.791,195.305,-110.174,169.572,44.635,158.442
C09756=1030.797,195.553,-110.199,169.575,44.633,158.442
C09757=1030.803,195.802,-110.223,169.579,44.631,158.442
C09758=1030.809,196.051,-110.248,169.583,44.630,158.442
C09759=1030.815,196.300,-110.272,169.586,44.628,158.442
C09760=1030.821,196.549,-110.296,169.590,44.625,158.442
C09761=1030.827,196.797,-110.320,169.594,44.624,158.442
C09762=1030.833,197.046,-110.345,169.596,44.622,158.441
C09763=1030.840,197.295,-110.369,169.600,44.620,158.442
C09764=1030.845,197.544,-110.393,169.604,44.618,158.441
C09765=1030.852,197.793,-110.418,169.607,44.617,158.441
C09766=1030.858,198.041,-110.443,169.611,44.615,158.441
C09767=1030.864,198.289,-110.467,169.615,44.613,158.441
C09768=1030.870,198.539,-110.491,169.618,44.611,158.441
C09769=1030.877,198.788,-110.515,169.621,44.610,158.441
C09770=1030.882,199.036,-110.540,169.625,44.608,158.441
C09771=1030.889,199.285,-110.564,169.629,44.606,158.441
C09772=1030.895,199.534,-110.589,169.632,44.605,158.441
C09773=1030.901,199.782,-110.613,169.636,44.603,158.441
C09774=1030.907,200.031,-110.638,169.640,44.601,158.441
C09775=1030.914,200.280,-110.662,169.643,44.599,158.441
C09776=1030.920,200.529,-110.687,169.647,44.597,158.441
C09777=1030.925,200.777,-110.711,169.651,44.596,158.441
C09778=1030.932,201.026,-110.737,169.653,44.594,158.441
C09779=1030.937,201.275,-110.761,169.657,44.593,158.441
C09780=1030.944,201.523,-110.786,169.661,44.591,158.441
C09781=1030.950,201.772,-110.810,169.665,44.589,158.441
C09782=1030.956,202.021,-110.836,169.668,44.587,158.441
C09783=1030.961,202.269,-110.860,169.672,44.586,158.441
C09784=1030.967,202.518,-110.885,169.676,44.585,158.441
C09785=1030.973,202.767,-110.910,169.679,44.583,158.441
C09786=1030.980,203.016,-110.935,169.682,44.581,158.441
C09787=1030.986,203.264,-110.960,169.686,44.580,158.441
C09788=1030.992,203.513,-110.984,169.690,44.578,158.441
C09789=1030.998,203.762,-111.010,169.694,44.576,158.441
C09790=1031.003,204.010,-111.034,169.698,44.575,158.441
C09791=1031.029,205.059,-111.139,170.049,44.679,158.497
C09792=1031.039,205.420,-111.177,170.053,44.677,158.497
C09793=1031.049,205.780,-111.215,170.057,44.676,158.497
C09794=1031.059,206.142,-111.254,170.061,44.675,158.497
C09795=1031.069,206.503,-111.291,170.064,44.673,158.497
C09796=1031.076,206.752,-111.318,170.067,44.673,158.497
C09797=1031.081,207.000,-111.344,170.069,44.672,158.497
C09798=1031.089,207.249,-111.371,170.072,44.671,158.497
C09799=1031.095,207.497,-111.397,170.075,44.671,158.497
C09800=1031.102,207.746,-111.423,170.078,44.669,158.497
C09801=1031.109,207.994,-111.449,170.080,44.669,158.497
C09802=1031.115,208.243,-111.476,170.083,44.668,158.497
C09803=1031.122,208.492,-111.503,170.086,44.667,158.498
C09804=1031.129,208.739,-111.530,170.089,44.666,158.498
C09805=1031.136,208.988,-111.556,170.091,44.665,158.498
C09806=1031.142,209.236,-111.583,170.094,44.665,158.498
C09807=1031.149,209.485,-111.609,170.097,44.664,158.498
C09808=1031.156,209.734,-111.635,170.099,44.663,158.498
C09809=1031.163,209.982,-111.662,170.102,44.662,158.498
C09810=1031.169,210.231,-111.689,170.105,44.662,158.498
C09811=1031.176,210.479,-111.715,170.108,44.660,158.498
C09812=1031.183,210.728,-111.741,170.110,44.660,158.498
C09813=1031.189,210.977,-111.768,170.113,44.659,158.499
C09814=1031.196,211.224,-111.795,170.115,44.658,158.499
C09815=1031.202,211.473,-111.822,170.118,44.657,158.499
C09816=1031.209,211.722,-111.848,170.120,44.657,158.499
C09817=1031.215,211.970,-111.875,170.124,44.656,158.499
C09818=1031.223,212.218,-111.902,170.127,44.656,158.499
C09819=1031.229,212.466,-111.928,170.129,44.654,158.499
C09820=1031.235,212.716,-111.955,170.131,44.654,158.499
C09821=1031.243,212.964,-111.982,170.134,44.653,158.499
C09822=1031.249,213.212,-112.009,170.137,44.653,158.499
C09823=1031.256,213.461,-112.035,170.140,44.651,158.499
C09824=1031.262,213.710,-112.062,170.142,44.651,158.500
C09825=1031.269,213.958,-112.088,170.145,44.650,158.500
C09826=1031.275,214.206,-112.116,170.148,44.650,158.500
C09827=1031.282,214.455,-112.143,170.151,44.648,158.500
C09828=1031.288,214.703,-112.169,170.153,44.648,158.500
C09829=1031.296,214.952,-112.196,170.156,44.647,158.500
C09830=1031.302,215.201,-112.223,170.159,44.647,158.500
C09831=1031.309,215.449,-112.250,170.162,44.645,158.500
C09832=1031.315,215.697,-112.277,170.165,44.645,158.500
C09833=1031.322,215.946,-112.304,170.167,44.644,158.501
C09834=1031.329,216.194,-112.331,170.170,44.644,158.501
C09835=1031.335,216.442,-112.357,170.173,44.643,158.501
C09836=1031.342,216.691,-112.384,170.176,44.642,158.501
C09837=1031.349,216.940,-112.411,170.179,44.641,158.501
C09838=1031.356,217.189,-112.438,170.181,44.641,158.501
C09839=1031.362,217.436,-112.465,170.184,44.640,158.501
C09840=1031.369,217.685,-112.492,170.187,44.639,158.501
C09841=1031.376,217.934,-112.519,170.190,44.638,158.501
C09842=1031.383,218.182,-112.546,170.193,44.638,158.502
C09843=1031.389,218.430,-112.572,170.195,44.637,158.502
C09844=1031.397,218.678,-112.600,170.198,44.636,158.502
C09845=1031.403,218.928,-112.627,170.201,44.635,158.502
C09846=1031.410,219.176,-112.654,170.204,44.635,158.502
C09847=1031.416,219.424,-112.680,170.207,44.634,158.502
C09848=1031.426,219.791,-112.721,170.211,44.633,158.502
C09849=1031.436,220.158,-112.761,170.215,44.632,158.503
C09850=1031.445,220.524,-112.801,170.219,44.631,158.503
C09851=1031.456,220.891,-112.842,170.223,44.631,158.503
C09852=1031.462,221.140,-112.869,170.226,44.630,158.503
C09853=1031.469,221.389,-112.896,170.229,44.629,158.503
C09854=1031.476,221.636,-112.923,170.232,44.628,158.503
C09855=1031.482,221.885,-112.950,170.234,44.628,158.503
C09856=1031.489,222.134,-112.978,170.237,44.627,158.504
C09857=1031.495,222.382,-113.006,170.240,44.626,158.504
C09858=1031.502,222.631,-113.032,170.243,44.626,158.504
C09859=1031.508,222.878,-113.059,170.246,44.625,158.504
C09860=1031.515,223.127,-113.087,170.249,44.624,158.504
C09861=1031.521,223.376,-113.114,170.251,44.624,158.504
C09862=1031.528,223.624,-113.142,170.254,44.623,158.504
C09863=1031.536,223.873,-113.169,170.257,44.623,158.505
C09864=1031.542,224.121,-113.197,170.260,44.622,158.505
C09865=1031.548,224.369,-113.223,170.263,44.621,158.505
C09866=1031.555,224.618,-113.251,170.266,44.621,158.505
C09867=1031.561,224.866,-113.279,170.268,44.620,158.505
C09868=1031.569,225.114,-113.306,170.271,44.620,158.505
C09869=1031.575,225.363,-113.333,170.274,44.619,158.505
C09870=1031.582,225.612,-113.361,170.277,44.618,158.506
C09871=1031.589,225.860,-113.389,170.281,44.618,158.506
C09872=1031.596,226.108,-113.416,170.284,44.617,158.506
C09873=1031.603,226.357,-113.443,170.287,44.616,158.506
C09874=1031.609,226.605,-113.471,170.289,44.616,158.506
C09875=1031.615,226.854,-113.498,170.292,44.615,158.506
C09876=1031.622,227.102,-113.526,170.295,44.615,158.506
C09877=1031.629,227.350,-113.553,170.298,44.614,158.507
C09878=1031.636,227.599,-113.580,170.301,44.613,158.507
C09879=1031.643,227.847,-113.608,170.304,44.613,158.507
C09880=1031.649,228.096,-113.636,170.307,44.612,158.507
C09881=1031.656,228.344,-113.664,170.310,44.612,158.507
C09882=1031.663,228.592,-113.691,170.312,44.611,158.507
C09883=1031.669,228.841,-113.719,170.315,44.611,158.507
C09884=1031.676,229.089,-113.747,170.318,44.610,158.508
C09885=1031.683,229.338,-113.774,170.321,44.609,158.508
C09886=1031.689,229.585,-113.802,170.324,44.609,158.508
C09887=1031.695,229.834,-113.830,170.327,44.608,158.508
C09888=1031.702,230.082,-113.857,170.330,44.607,158.508
C09889=1031.709,230.331,-113.885,170.333,44.607,158.509
C09890=1031.715,230.579,-113.913,170.335,44.607,158.509
C09891=1031.722,230.828,-113.941,170.338,44.606,158.509
C09892=1031.729,231.076,-113.968,170.342,44.606,158.509
C09893=1031.736,231.325,-113.996,170.345,44.605,158.509
C09894=1031.742,231.573,-114.025,170.348,44.604,158.509
C09895=1031.748,231.821,-114.053,170.351,44.604,158.509
C09896=1031.755,232.070,-114.080,170.354,44.604,158.510
C09897=1031.762,232.318,-114.108,170.357,44.603,158.510
C09898=1031.769,232.566,-114.136,170.360,44.602,158.510
C09899=1031.775,232.815,-114.164,170.362,44.602,158.510
C09900=1031.781,233.063,-114.193,170.365,44.601,158.510
C09901=1031.788,233.311,-114.220,170.368,44.601,158.510
C09902=1031.795,233.560,-114.248,170.371,44.601,158.511
C09903=1031.801,233.808,-114.276,170.374,44.600,158.511
C09904=1031.811,234.167,-114.317,170.378,44.599,158.511
C09905=1031.821,234.527,-114.357,170.383,44.598,158.511
C09906=1031.831,234.886,-114.398,170.388,44.598,158.512
C09907=1031.840,235.245,-114.439,170.392,44.597,158.512
C09908=1031.847,235.493,-114.466,170.395,44.597,158.512
C09909=1031.853,235.742,-114.494,170.398,44.597,158.512
C09910=1031.860,235.989,-114.523,170.401,44.596,158.513
C09911=1031.866,236.238,-114.551,170.404,44.595,158.513
C09912=1031.873,236.487,-114.579,170.407,44.595,158.513
C09913=1031.880,236.734,-114.607,170.410,44.594,158.513
C09914=1031.887,236.984,-114.635,170.414,44.594,158.513
C09915=1031.894,237.232,-114.663,170.417,44.593,158.513
C09916=1031.900,237.480,-114.692,170.419,44.593,158.514
C09917=1031.907,237.729,-114.720,170.422,44.592,158.514
C09918=1031.914,237.976,-114.748,170.425,44.592,158.514
C09919=1031.920,238.225,-114.776,170.428,44.592,158.514
C09920=1031.926,238.474,-114.804,170.431,44.591,158.514
C09921=1031.933,238.721,-114.833,170.434,44.591,158.515
C09922=1031.940,238.970,-114.860,170.437,44.590,158.515
C09923=1031.946,239.218,-114.889,170.440,44.590,158.515
C09924=1031.954,239.467,-114.918,170.443,44.589,158.515
C09925=1031.961,239.715,-114.946,170.447,44.589,158.515
C09926=1031.967,239.963,-114.974,170.450,44.588,158.516
C09927=1031.973,240.212,-115.003,170.453,44.588,158.516
C09928=1031.980,240.460,-115.030,170.456,44.588,158.516
C09929=1031.986,240.708,-115.060,170.459,44.587,158.516
C09930=1031.993,240.956,-115.088,170.462,44.587,158.516
C09931=1032.000,241.205,-115.117,170.465,44.586,158.517
C09932=1032.007,241.453,-115.145,170.468,44.586,158.517
C09933=1032.013,241.701,-115.174,170.472,44.586,158.517
C09934=1032.020,241.950,-115.202,170.475,44.585,158.517
C09935=1032.026,242.198,-115.231,170.478,44.585,158.518
C09936=1032.033,242.446,-115.259,170.481,44.585,158.518
C09937=1032.039,242.694,-115.288,170.484,44.584,158.518
C09938=1032.047,242.943,-115.316,170.487,44.584,158.518
C09939=1032.053,243.191,-115.346,170.490,44.583,158.518
C09940=1032.060,243.440,-115.373,170.494,44.583,158.519
C09941=1032.066,243.688,-115.402,170.497,44.583,158.519
C09942=1032.073,243.936,-115.431,170.500,44.583,158.519
C09943=1032.080,244.184,-115.460,170.503,44.582,158.519
C09944=1032.086,244.433,-115.488,170.506,44.581,158.519
C09945=1032.093,244.681,-115.517,170.509,44.581,158.520
C09946=1032.099,244.929,-115.546,170.513,44.581,158.520
C09947=1032.105,245.177,-115.575,170.516,44.581,158.520
C09948=1032.112,245.425,-115.603,170.519,44.581,158.520
C09949=1032.119,245.674,-115.633,170.521,44.580,158.521
C09950=1032.125,245.922,-115.662,170.524,44.580,158.521
C09951=1032.131,246.170,-115.691,170.527,44.580,158.521
C09952=1032.138,246.418,-115.720,170.531,44.580,158.521
C09953=1032.145,246.666,-115.748,170.534,44.580,158.522
C09954=1032.151,246.915,-115.778,170.537,44.579,158.522
C09955=1032.157,247.164,-115.806,170.540,44.579,158.522
C09956=1032.164,247.412,-115.835,170.543,44.578,158.522
C09957=1032.171,247.660,-115.864,170.547,44.578,158.523
C09958=1032.177,247.908,-115.893,170.550,44.578,158.523
C09959=1032.184,248.157,-115.922,170.553,44.578,158.523
C09960=1032.193,248.509,-115.963,170.558,44.577,158.523
C09961=1032.202,248.863,-116.005,170.562,44.577,158.524
C09962=1032.211,249.216,-116.047,170.567,44.577,158.524
C09963=1032.221,249.569,-116.088,170.572,44.576,158.525
C09964=1032.228,249.817,-116.117,170.575,44.576,158.525
C09965=1032.234,250.066,-116.146,170.578,44.576,158.525
C09966=1032.242,250.314,-116.175,170.582,44.576,158.525
C09967=1032.248,250.562,-116.204,170.585,44.575,158.525
C09968=1032.254,250.810,-116.233,170.588,44.575,158.526
C09969=1032.261,251.059,-116.263,170.591,44.575,158.526
C09970=1032.267,251.307,-116.292,170.594,44.575,158.526
C09971=1032.274,251.554,-116.321,170.598,44.574,158.527
C09972=1032.281,251.803,-116.350,170.601,44.574,158.527
C09973=1032.288,252.051,-116.379,170.604,44.574,158.527
C09974=1032.294,252.300,-116.408,170.607,44.574,158.527
C09975=1032.301,252.548,-116.438,170.610,44.574,158.528
C09976=1032.307,252.796,-116.467,170.613,44.573,158.528
C09977=1032.314,253.044,-116.496,170.617,44.573,158.528
C09978=1032.321,253.293,-116.525,170.620,44.573,158.528
C09979=1032.327,253.541,-116.554,170.624,44.572,158.529
C09980=1032.334,253.790,-116.584,170.627,44.572,158.529
C09981=1032.341,254.037,-116.614,170.631,44.572,158.529
C09982=1032.348,254.285,-116.642,170.634,44.572,158.529
C09983=1032.355,254.534,-116.671,170.637,44.572,158.530
C09984=1032.361,254.781,-116.701,170.640,44.572,158.530
C09985=1032.368,255.030,-116.731,170.643,44.571,158.530
C09986=1032.374,255.278,-116.760,170.647,44.571,158.530
C09987=1032.381,255.526,-116.790,170.650,44.571,158.531
C09988=1032.388,255.774,-116.818,170.654,44.570,158.531
C09989=1032.395,256.023,-116.848,170.657,44.570,158.531
C09990=1032.402,256.271,-116.877,170.660,44.570,158.532
C09991=1032.408,256.519,-116.906,170.664,44.570,158.532
C09992=1032.415,256.768,-116.936,170.667,44.570,158.532
C09993=1032.421,257.015,-116.965,170.670,44.569,158.532
C09994=1032.428,257.264,-116.995,170.673,44.569,158.533
C09995=1032.436,257.511,-117.024,170.677,44.569,158.533
C09996=1032.442,257.760,-117.053,170.681,44.569,158.533
//INST
///DATE 2021/06/17 10:58
///ATTR SC,RW,RJ
////FRAME ROBOT
///GROUP1 RB1
NOP
MOVL C00000 V=800.0 PL=0
MOVL C00001 V=800.0 PL=0
MOVL C00002 V=800.0 PL=0
MOVL C00003 V=800.0 PL=0
MOVL C00004 V=800.0 PL=0
MOVL C00005 V=800.0 PL=0
MOVL C00006 V=800.0 PL=0
MOVL C00007 V=800.0 PL=0
MOVL C00008 V=800.0 PL=0
MOVL C00009 V=800.0 PL=0
MOVL C00010 V=800.0 PL=0
MOVL C00011 V=800.0 PL=0
MOVL C00012 V=800.0 PL=0
MOVL C00013 V=800.0 PL=0
MOVL C00014 V=800.0 PL=0
MOVL C00015 V=800.0 PL=0
MOVL C00016 V=800.0 PL=0
MOVL C00017 V=800.0 PL=0
MOVL C00018 V=800.0 PL=0
MOVL C00019 V=800.0 PL=0
MOVL C00020 V=800.0 PL=0
MOVL C00021 V=800.0 PL=0
MOVL C00022 V=800.0 PL=0
MOVL C00023 V=800.0 PL=0
MOVL C00024 V=800.0 PL=0
MOVL C00025 V=800.0 PL=0
MOVL C00026 V=800.0 PL=0
MOVL C00027 V=800.0 PL=0
MOVL C00028 V=800.0 PL=0
MOVL C00029 V=800.0 PL=0
MOVL C00030 V=800.0 PL=0
MOVL C00031 V=800.0 PL=0
MOVL C00032 V=800.0 PL=0
MOVL C00033 V=800.0 PL=0
MOVL C00034 V=800.0 PL=0
MOVL C00035 V=800.0 PL=0
MOVL C00036 V=800.0 PL=0
MOVL C00037 V=800.0 PL=0
MOVL C00038 V=800.0 PL=0
MOVL C00039 V=800.0 PL=0
MOVL C00040 V=800.0 PL=0
MOVL C00041 V=800.0 PL=0
MOVL C00042 V=800.0 PL=0
MOVL C00043 V=800.0 PL=0
MOVL C00044 V=800.0 PL=0
MOVL C00045 V=800.0 PL=0
MOVL C00046 V=800.0 PL=0
MOVL C00047 V=800.0 PL=0
MOVL C00048 V=800.0 PL=0
MOVL C00049 V=800.0 PL=0
MOVL C00050 V=800.0 PL=0
MOVL C00051 V=800.0 PL=0
MOVL C00052 V=800.0 PL=0
MOVL C00053 V=800.0 PL=0
MOVL C00054 V=800.0 PL=0
MOVL C00055 V=800.0 PL=0
MOVL C00056 V=800.0 PL=0
MOVL C00057 V=800.0 PL=0
MOVL C00058 V=800.0 PL=0
MOVL C00059 V=800.0 PL=0
MOVL C00060 V=800.0 PL=0
MOVL C00061 V=800.0 PL=0
MOVL C00062 V=800.0 PL=0
MOVL C00063 V=800.0 PL=0
MOVL C00064 V=800.0 PL=0
MOVL C00065 V=800.0 PL=0
MOVL C00066 V=800.0 PL=0
MOVL C00067 V=800.0 PL=0
MOVL C00068 V=800.0 PL=0
MOVL C00069 V=800.0 PL=0
MOVL C00070 V=800.0 PL=0
MOVL C00071 V=800.0 PL=0
MOVL C00072 V=800.0 PL=0
MOVL C00073 V=800.0 PL=0
MOVL C00074 V=800.0 PL=0
MOVL C00075 V=800.0 PL=0
MOVL C00076 V=800.0 PL=0
MOVL C00077 V=800.0 PL=0
MOVL C00078 V=800.0 PL=0
MOVL C00079 V=800.0 PL=0
MOVL C00080 V=800.0 PL=0
MOVL C00081 V=800.0 PL=0
MOVL C00082 V=800.0 PL=0
MOVL C00083 V=800.0 PL=0
MOVL C00084 V=800.0 PL=0
MOVL C00085 V=800.0 PL=0
MOVL C00086 V=800.0 PL=0
MOVL C00087 V=800.0 PL=0
MOVL C00088 V=800.0 PL=0
MOVL C00089 V=800.0 PL=0
MOVL C00090 V=800.0 PL=0
MOVL C00091 V=800.0 PL=0
MOVL C00092 V=800.0 PL=0
MOVL C00093 V=800.0 PL=0
MOVL C00094 V=800.0 PL=0
MOVL C00095 V=800.0 PL=0
MOVL C00096 V=800.0 PL=0
MOVL C00097 V=800.0 PL=0
MOVL C00098 V=800.0 PL=0
MOVL C00099 V=800.0 PL=0
MOVL C00100 V=800.0 PL=0
MOVL C00101 V=800.0 PL=0
MOVL C00102 V=800.0 PL=0
MOVL C00103 V=800.0 PL=0
MOVL C00104 V=800.0 PL=0
MOVL C00105 V=800.0 PL=0
MOVL C00106 V=800.0 PL=0
MOVL C00107 V=800.0 PL=0
MOVL C00108 V=800.0 PL=0
MOVL C00109 V=800.0 PL=0
MOVL C00110 V=800.0 PL=0
MOVL C00111 V=800.0 PL=0
MOVL C00112 V=800.0 PL=0
MOVL C00113 V=800.0 PL=0
MOVL C00114 V=800.0 PL=0
MOVL C00115 V=800.0 PL=0
MOVL C00116 V=800.0 PL=0
MOVL C00117 V=800.0 PL=0
MOVL C00118 V=800.0 PL=0
MOVL C00119 V=800.0 PL=0
MOVL C00120 V=800.0 PL=0
MOVL C00121 V=800.0 PL=0
MOVL C00122 V=800.0 PL=0
MOVL C00123 V=800.0 PL=0
MOVL C00124 V=800.0 PL=0
MOVL C00125 V=800.0 PL=0
MOVL C00126 V=800.0 PL=0
MOVL C00127 V=800.0 PL=0
MOVL C00128 V=800.0 PL=0
MOVL C00129 V=800.0 PL=0
MOVL C00130 V=800.0 PL=0
MOVL C00131 V=800.0 PL=0
MOVL C00132 V=800.0 PL=0
MOVL C00133 V=800.0 PL=0
MOVL C00134 V=800.0 PL=0
MOVL C00135 V=800.0 PL=0
MOVL C00136 V=800.0 PL=0
MOVL C00137 V=800.0 PL=0
MOVL C00138 V=800.0 PL=0
MOVL C00139 V=800.0 PL=0
MOVL C00140 V=800.0 PL=0
MOVL C00141 V=800.0 PL=0
MOVL C00142 V=800.0 PL=0
MOVL C00143 V=800.0 PL=0
MOVL C00144 V=800.0 PL=0
MOVL C00145 V=800.0 PL=0
MOVL C00146 V=800.0 PL=0
MOVL C00147 V=800.0 PL=0
MOVL C00148 V=800.0 PL=0
MOVL C00149 V=800.0 PL=0
MOVL C00150 V=800.0 PL=0
MOVL C00151 V=800.0 PL=0
MOVL C00152 V=800.0 PL=0
MOVL C00153 V=800.0 PL=0
MOVL C00154 V=800.0 PL=0
MOVL C00155 V=800.0 PL=0
MOVL C00156 V=800.0 PL=0
MOVL C00157 V=800.0 PL=0
MOVL C00158 V=800.0 PL=0
MOVL C00159 V=800.0 PL=0
MOVL C00160 V=800.0 PL=0
MOVL C00161 V=800.0 PL=0
MOVL C00162 V=800.0 PL=0
MOVL C00163 V=800.0 PL=0
MOVL C00164 V=800.0 PL=0
MOVL C00165 V=800.0 PL=0
MOVL C00166 V=800.0 PL=0
MOVL C00167 V=800.0 PL=0
MOVL C00168 V=800.0 PL=0
MOVL C00169 V=800.0 PL=0
MOVL C00170 V=800.0 PL=0
MOVL C00171 V=800.0 PL=0
MOVL C00172 V=800.0 PL=0
MOVL C00173 V=800.0 PL=0
MOVL C00174 V=800.0 PL=0
MOVL C00175 V=800.0 PL=0
MOVL C00176 V=800.0 PL=0
MOVL C00177 V=800.0 PL=0
MOVL C00178 V=800.0 PL=0
MOVL C00179 V=800.0 PL=0
MOVL C00180 V=800.0 PL=0
MOVL C00181 V=800.0 PL=0
MOVL C00182 V=800.0 PL=0
MOVL C00183 V=800.0 PL=0
MOVL C00184 V=800.0 PL=0
MOVL C00185 V=800.0 PL=0
MOVL C00186 V=800.0 PL=0
MOVL C00187 V=800.0 PL=0
MOVL C00188 V=800.0 PL=0
MOVL C00189 V=800.0 PL=0
MOVL C00190 V=800.0 PL=0
MOVL C00191 V=800.0 PL=0
MOVL C00192 V=800.0 PL=0
MOVL C00193 V=800.0 PL=0
MOVL C00194 V=800.0 PL=0
MOVL C00195 V=800.0 PL=0
MOVL C00196 V=800.0 PL=0
MOVL C00197 V=800.0 PL=0
MOVL C00198 V=800.0 PL=0
MOVL C00199 V=800.0 PL=0
MOVL C00200 V=800.0 PL=0
MOVL C00201 V=800.0 PL=0
MOVL C00202 V=800.0 PL=0
MOVL C00203 V=800.0 PL=0
MOVL C00204 V=800.0 PL=0
MOVL C00205 V=800.0 PL=0
MOVL C00206 V=800.0 PL=0
MOVL C00207 V=800.0 PL=0
MOVL C00208 V=800.0 PL=0
MOVL C00209 V=800.0 PL=0
MOVL C00210 V=800.0 PL=0
MOVL C00211 V=800.0 PL=0
MOVL C00212 V=800.0 PL=0
MOVL C00213 V=800.0 PL=0
MOVL C00214 V=800.0 PL=0
MOVL C00215 V=800.0 PL=0
MOVL C00216 V=800.0 PL=0
MOVL C00217 V=800.0 PL=0
MOVL C00218 V=800.0 PL=0
MOVL C00219 V=800.0 PL=0
MOVL C00220 V=800.0 PL=0
MOVL C00221 V=800.0 PL=0
MOVL C00222 V=800.0 PL=0
MOVL C00223 V=800.0 PL=0
MOVL C00224 V=800.0 PL=0
MOVL C00225 V=800.0 PL=0
MOVL C00226 V=800.0 PL=0
MOVL C00227 V=800.0 PL=0
MOVL C00228 V=800.0 PL=0
MOVL C00229 V=800.0 PL=0
MOVL C00230 V=800.0 PL=0
MOVL C00231 V=800.0 PL=0
MOVL C00232 V=800.0 PL=0
MOVL C00233 V=800.0 PL=0
MOVL C00234 V=800.0 PL=0
MOVL C00235 V=800.0 PL=0
MOVL C00236 V=800.0 PL=0
MOVL C00237 V=800.0 PL=0
MOVL C00238 V=800.0 PL=0
MOVL C00239 V=800.0 PL=0
MOVL C00240 V=800.0 PL=0
MOVL C00241 V=800.0 PL=0
MOVL C00242 V=800.0 PL=0
MOVL C00243 V=800.0 PL=0
MOVL C00244 V=800.0 PL=0
MOVL C00245 V=800.0 PL=0
MOVL C00246 V=800.0 PL=0
MOVL C00247 V=800.0 PL=0
MOVL C00248 V=800.0 PL=0
MOVL C00249 V=800.0 PL=0
MOVL C00250 V=800.0 PL=0
MOVL C00251 V=800.0 PL=0
MOVL C00252 V=800.0 PL=0
MOVL C00253 V=800.0 PL=0
MOVL C00254 V=800.0 PL=0
MOVL C00255 V=800.0 PL=0
MOVL C00256 V=800.0 PL=0
MOVL C00257 V=800.0 PL=0
MOVL C00258 V=800.0 PL=0
MOVL C00259 V=800.0 PL=0
MOVL C00260 V=800.0 PL=0
MOVL C00261 V=800.0 PL=0
MOVL C00262 V=800.0 PL=0
MOVL C00263 V=800.0 PL=0
MOVL C00264 V=800.0 PL=0
MOVL C00265 V=800.0 PL=0
MOVL C00266 V=800.0 PL=0
MOVL C00267 V=800.0 PL=0
MOVL C00268 V=800.0 PL=0
MOVL C00269 V=800.0 PL=0
MOVL C00270 V=800.0 PL=0
MOVL C00271 V=800.0 PL=0
MOVL C00272 V=800.0 PL=0
MOVL C00273 V=800.0 PL=0
MOVL C00274 V=800.0 PL=0
MOVL C00275 V=800.0 PL=0
MOVL C00276 V=800.0 PL=0
MOVL C00277 V=800.0 PL=0
MOVL C00278 V=800.0 PL=0
MOVL C00279 V=800.0 PL=0
MOVL C00280 V=800.0 PL=0
MOVL C00281 V=800.0 PL=0
MOVL C00282 V=800.0 PL=0
MOVL C00283 V=800.0 PL=0
MOVL C00284 V=800.0 PL=0
MOVL C00285 V=800.0 PL=0
MOVL C00286 V=800.0 PL=0
MOVL C00287 V=800.0 PL=0
MOVL C00288 V=800.0 PL=0
MOVL C00289 V=800.0 PL=0
MOVL C00290 V=800.0 PL=0
MOVL C00291 V=800.0 PL=0
MOVL C00292 V=800.0 PL=0
MOVL C00293 V=800.0 PL=0
MOVL C00294 V=800.0 PL=0
MOVL C00295 V=800.0 PL=0
MOVL C00296 V=800.0 PL=0
MOVL C00297 V=800.0 PL=0
MOVL C00298 V=800.0 PL=0
MOVL C00299 V=800.0 PL=0
MOVL C00300 V=800.0 PL=0
MOVL C00301 V=800.0 PL=0
MOVL C00302 V=800.0 PL=0
MOVL C00303 V=800.0 PL=0
MOVL C00304 V=800.0 PL=0
MOVL C00305 V=800.0 PL=0
MOVL C00306 V=800.0 PL=0
MOVL C00307 V=800.0 PL=0
MOVL C00308 V=800.0 PL=0
MOVL C00309 V=800.0 PL=0
MOVL C00310 V=800.0 PL=0
MOVL C00311 V=800.0 PL=0
MOVL C00312 V=800.0 PL=0
MOVL C00313 V=800.0 PL=0
MOVL C00314 V=800.0 PL=0
MOVL C00315 V=800.0 PL=0
MOVL C00316 V=800.0 PL=0
MOVL C00317 V=800.0 PL=0
MOVL C00318 V=800.0 PL=0
MOVL C00319 V=800.0 PL=0
MOVL C00320 V=800.0 PL=0
MOVL C00321 V=800.0 PL=0
MOVL C00322 V=800.0 PL=0
MOVL C00323 V=800.0 PL=0
MOVL C00324 V=800.0 PL=0
MOVL C00325 V=800.0 PL=0
MOVL C00326 V=800.0 PL=0
MOVL C00327 V=800.0 PL=0
MOVL C00328 V=800.0 PL=0
MOVL C00329 V=800.0 PL=0
MOVL C00330 V=800.0 PL=0
MOVL C00331 V=800.0 PL=0
MOVL C00332 V=800.0 PL=0
MOVL C00333 V=800.0 PL=0
MOVL C00334 V=800.0 PL=0
MOVL C00335 V=800.0 PL=0
MOVL C00336 V=800.0 PL=0
MOVL C00337 V=800.0 PL=0
MOVL C00338 V=800.0 PL=0
MOVL C00339 V=800.0 PL=0
MOVL C00340 V=800.0 PL=0
MOVL C00341 V=800.0 PL=0
MOVL C00342 V=800.0 PL=0
MOVL C00343 V=800.0 PL=0
MOVL C00344 V=800.0 PL=0
MOVL C00345 V=800.0 PL=0
MOVL C00346 V=800.0 PL=0
MOVL C00347 V=800.0 PL=0
MOVL C00348 V=800.0 PL=0
MOVL C00349 V=800.0 PL=0
MOVL C00350 V=800.0 PL=0
MOVL C00351 V=800.0 PL=0
MOVL C00352 V=800.0 PL=0
MOVL C00353 V=800.0 PL=0
MOVL C00354 V=800.0 PL=0
MOVL C00355 V=800.0 PL=0
MOVL C00356 V=800.0 PL=0
MOVL C00357 V=800.0 PL=0
MOVL C00358 V=800.0 PL=0
MOVL C00359 V=800.0 PL=0
MOVL C00360 V=800.0 PL=0
MOVL C00361 V=800.0 PL=0
MOVL C00362 V=800.0 PL=0
MOVL C00363 V=800.0 PL=0
MOVL C00364 V=800.0 PL=0
MOVL C00365 V=800.0 PL=0
MOVL C00366 V=800.0 PL=0
MOVL C00367 V=800.0 PL=0
MOVL C00368 V=800.0 PL=0
MOVL C00369 V=800.0 PL=0
MOVL C00370 V=800.0 PL=0
MOVL C00371 V=800.0 PL=0
MOVL C00372 V=800.0 PL=0
MOVL C00373 V=800.0 PL=0
MOVL C00374 V=800.0 PL=0
MOVL C00375 V=800.0 PL=0
MOVL C00376 V=800.0 PL=0
MOVL C00377 V=800.0 PL=0
MOVL C00378 V=800.0 PL=0
MOVL C00379 V=800.0 PL=0
MOVL C00380 V=800.0 PL=0
MOVL C00381 V=800.0 PL=0
MOVL C00382 V=800.0 PL=0
MOVL C00383 V=800.0 PL=0
MOVL C00384 V=800.0 PL=0
MOVL C00385 V=800.0 PL=0
MOVL C00386 V=800.0 PL=0
MOVL C00387 V=800.0 PL=0
MOVL C00388 V=800.0 PL=0
MOVL C00389 V=800.0 PL=0
MOVL C00390 V=800.0 PL=0
MOVL C00391 V=800.0 PL=0
MOVL C00392 V=800.0 PL=0
MOVL C00393 V=800.0 PL=0
MOVL C00394 V=800.0 PL=0
MOVL C00395 V=800.0 PL=0
MOVL C00396 V=800.0 PL=0
MOVL C00397 V=800.0 PL=0
MOVL C00398 V=800.0 PL=0
MOVL C00399 V=800.0 PL=0
MOVL C00400 V=800.0 PL=0
MOVL C00401 V=800.0 PL=0
MOVL C00402 V=800.0 PL=0
MOVL C00403 V=800.0 PL=0
MOVL C00404 V=800.0 PL=0
MOVL C00405 V=800.0 PL=0
MOVL C00406 V=800.0 PL=0
MOVL C00407 V=800.0 PL=0
MOVL C00408 V=800.0 PL=0
MOVL C00409 V=800.0 PL=0
MOVL C00410 V=800.0 PL=0
MOVL C00411 V=800.0 PL=0
MOVL C00412 V=800.0 PL=0
MOVL C00413 V=800.0 PL=0
MOVL C00414 V=800.0 PL=0
MOVL C00415 V=800.0 PL=0
MOVL C00416 V=800.0 PL=0
MOVL C00417 V=800.0 PL=0
MOVL C00418 V=800.0 PL=0
MOVL C00419 V=800.0 PL=0
MOVL C00420 V=800.0 PL=0
MOVL C00421 V=800.0 PL=0
MOVL C00422 V=800.0 PL=0
MOVL C00423 V=800.0 PL=0
MOVL C00424 V=800.0 PL=0
MOVL C00425 V=800.0 PL=0
MOVL C00426 V=800.0 PL=0
MOVL C00427 V=800.0 PL=0
MOVL C00428 V=800.0 PL=0
MOVL C00429 V=800.0 PL=0
MOVL C00430 V=800.0 PL=0
MOVL C00431 V=800.0 PL=0
MOVL C00432 V=800.0 PL=0
MOVL C00433 V=800.0 PL=0
MOVL C00434 V=800.0 PL=0
MOVL C00435 V=800.0 PL=0
MOVL C00436 V=800.0 PL=0
MOVL C00437 V=800.0 PL=0
MOVL C00438 V=800.0 PL=0
MOVL C00439 V=800.0 PL=0
MOVL C00440 V=800.0 PL=0
MOVL C00441 V=800.0 PL=0
MOVL C00442 V=800.0 PL=0
MOVL C00443 V=800.0 PL=0
MOVL C00444 V=800.0 PL=0
MOVL C00445 V=800.0 PL=0
MOVL C00446 V=800.0 PL=0
MOVL C00447 V=800.0 PL=0
MOVL C00448 V=800.0 PL=0
MOVL C00449 V=800.0 PL=0
MOVL C00450 V=800.0 PL=0
MOVL C00451 V=800.0 PL=0
MOVL C00452 V=800.0 PL=0
MOVL C00453 V=800.0 PL=0
MOVL C00454 V=800.0 PL=0
MOVL C00455 V=800.0 PL=0
MOVL C00456 V=800.0 PL=0
MOVL C00457 V=800.0 PL=0
MOVL C00458 V=800.0 PL=0
MOVL C00459 V=800.0 PL=0
MOVL C00460 V=800.0 PL=0
MOVL C00461 V=800.0 PL=0
MOVL C00462 V=800.0 PL=0
MOVL C00463 V=800.0 PL=0
MOVL C00464 V=800.0 PL=0
MOVL C00465 V=800.0 PL=0
MOVL C00466 V=800.0 PL=0
MOVL C00467 V=800.0 PL=0
MOVL C00468 V=800.0 PL=0
MOVL C00469 V=800.0 PL=0
MOVL C00470 V=800.0 PL=0
MOVL C00471 V=800.0 PL=0
MOVL C00472 V=800.0 PL=0
MOVL C00473 V=800.0 PL=0
MOVL C00474 V=800.0 PL=0
MOVL C00475 V=800.0 PL=0
MOVL C00476 V=800.0 PL=0
MOVL C00477 V=800.0 PL=0
MOVL C00478 V=800.0 PL=0
MOVL C00479 V=800.0 PL=0
MOVL C00480 V=800.0 PL=0
MOVL C00481 V=800.0 PL=0
MOVL C00482 V=800.0 PL=0
MOVL C00483 V=800.0 PL=0
MOVL C00484 V=800.0 PL=0
MOVL C00485 V=800.0 PL=0
MOVL C00486 V=800.0 PL=0
MOVL C00487 V=800.0 PL=0
MOVL C00488 V=800.0 PL=0
MOVL C00489 V=800.0 PL=0
MOVL C00490 V=800.0 PL=0
MOVL C00491 V=800.0 PL=0
MOVL C00492 V=800.0 PL=0
MOVL C00493 V=800.0 PL=0
MOVL C00494 V=800.0 PL=0
MOVL C00495 V=800.0 PL=0
MOVL C00496 V=800.0 PL=0
MOVL C00497 V=800.0 PL=0
MOVL C00498 V=800.0 PL=0
MOVL C00499 V=800.0 PL=0
MOVL C00500 V=800.0 PL=0
MOVL C00501 V=800.0 PL=0
MOVL C00502 V=800.0 PL=0
MOVL C00503 V=800.0 PL=0
MOVL C00504 V=800.0 PL=0
MOVL C00505 V=800.0 PL=0
MOVL C00506 V=800.0 PL=0
MOVL C00507 V=800.0 PL=0
MOVL C00508 V=800.0 PL=0
MOVL C00509 V=800.0 PL=0
MOVL C00510 V=800.0 PL=0
MOVL C00511 V=800.0 PL=0
MOVL C00512 V=800.0 PL=0
MOVL C00513 V=800.0 PL=0
MOVL C00514 V=800.0 PL=0
MOVL C00515 V=800.0 PL=0
MOVL C00516 V=800.0 PL=0
MOVL C00517 V=800.0 PL=0
MOVL C00518 V=800.0 PL=0
MOVL C00519 V=800.0 PL=0
MOVL C00520 V=800.0 PL=0
MOVL C00521 V=800.0 PL=0
MOVL C00522 V=800.0 PL=0
MOVL C00523 V=800.0 PL=0
MOVL C00524 V=800.0 PL=0
MOVL C00525 V=800.0 PL=0
MOVL C00526 V=800.0 PL=0
MOVL C00527 V=800.0 PL=0
MOVL C00528 V=800.0 PL=0
MOVL C00529 V=800.0 PL=0
MOVL C00530 V=800.0 PL=0
MOVL C00531 V=800.0 PL=0
MOVL C00532 V=800.0 PL=0
MOVL C00533 V=800.0 PL=0
MOVL C00534 V=800.0 PL=0
MOVL C00535 V=800.0 PL=0
MOVL C00536 V=800.0 PL=0
MOVL C00537 V=800.0 PL=0
MOVL C00538 V=800.0 PL=0
MOVL C00539 V=800.0 PL=0
MOVL C00540 V=800.0 PL=0
MOVL C00541 V=800.0 PL=0
MOVL C00542 V=800.0 PL=0
MOVL C00543 V=800.0 PL=0
MOVL C00544 V=800.0 PL=0
MOVL C00545 V=800.0 PL=0
MOVL C00546 V=800.0 PL=0
MOVL C00547 V=800.0 PL=0
MOVL C00548 V=800.0 PL=0
MOVL C00549 V=800.0 PL=0
MOVL C00550 V=800.0 PL=0
MOVL C00551 V=800.0 PL=0
MOVL C00552 V=800.0 PL=0
MOVL C00553 V=800.0 PL=0
MOVL C00554 V=800.0 PL=0
MOVL C00555 V=800.0 PL=0
MOVL C00556 V=800.0 PL=0
MOVL C00557 V=800.0 PL=0
MOVL C00558 V=800.0 PL=0
MOVL C00559 V=800.0 PL=0
MOVL C00560 V=800.0 PL=0
MOVL C00561 V=800.0 PL=0
MOVL C00562 V=800.0 PL=0
MOVL C00563 V=800.0 PL=0
MOVL C00564 V=800.0 PL=0
MOVL C00565 V=800.0 PL=0
MOVL C00566 V=800.0 PL=0
MOVL C00567 V=800.0 PL=0
MOVL C00568 V=800.0 PL=0
MOVL C00569 V=800.0 PL=0
MOVL C00570 V=800.0 PL=0
MOVL C00571 V=800.0 PL=0
MOVL C00572 V=800.0 PL=0
MOVL C00573 V=800.0 PL=0
MOVL C00574 V=800.0 PL=0
MOVL C00575 V=800.0 PL=0
MOVL C00576 V=800.0 PL=0
MOVL C00577 V=800.0 PL=0
MOVL C00578 V=800.0 PL=0
MOVL C00579 V=800.0 PL=0
MOVL C00580 V=800.0 PL=0
MOVL C00581 V=800.0 PL=0
MOVL C00582 V=800.0 PL=0
MOVL C00583 V=800.0 PL=0
MOVL C00584 V=800.0 PL=0
MOVL C00585 V=800.0 PL=0
MOVL C00586 V=800.0 PL=0
MOVL C00587 V=800.0 PL=0
MOVL C00588 V=800.0 PL=0
MOVL C00589 V=800.0 PL=0
MOVL C00590 V=800.0 PL=0
MOVL C00591 V=800.0 PL=0
MOVL C00592 V=800.0 PL=0
MOVL C00593 V=800.0 PL=0
MOVL C00594 V=800.0 PL=0
MOVL C00595 V=800.0 PL=0
MOVL C00596 V=800.0 PL=0
MOVL C00597 V=800.0 PL=0
MOVL C00598 V=800.0 PL=0
MOVL C00599 V=800.0 PL=0
MOVL C00600 V=800.0 PL=0
MOVL C00601 V=800.0 PL=0
MOVL C00602 V=800.0 PL=0
MOVL C00603 V=800.0 PL=0
MOVL C00604 V=800.0 PL=0
MOVL C00605 V=800.0 PL=0
MOVL C00606 V=800.0 PL=0
MOVL C00607 V=800.0 PL=0
MOVL C00608 V=800.0 PL=0
MOVL C00609 V=800.0 PL=0
MOVL C00610 V=800.0 PL=0
MOVL C00611 V=800.0 PL=0
MOVL C00612 V=800.0 PL=0
MOVL C00613 V=800.0 PL=0
MOVL C00614 V=800.0 PL=0
MOVL C00615 V=800.0 PL=0
MOVL C00616 V=800.0 PL=0
MOVL C00617 V=800.0 PL=0
MOVL C00618 V=800.0 PL=0
MOVL C00619 V=800.0 PL=0
MOVL C00620 V=800.0 PL=0
MOVL C00621 V=800.0 PL=0
MOVL C00622 V=800.0 PL=0
MOVL C00623 V=800.0 PL=0
MOVL C00624 V=800.0 PL=0
MOVL C00625 V=800.0 PL=0
MOVL C00626 V=800.0 PL=0
MOVL C00627 V=800.0 PL=0
MOVL C00628 V=800.0 PL=0
MOVL C00629 V=800.0 PL=0
MOVL C00630 V=800.0 PL=0
MOVL C00631 V=800.0 PL=0
MOVL C00632 V=800.0 PL=0
MOVL C00633 V=800.0 PL=0
MOVL C00634 V=800.0 PL=0
MOVL C00635 V=800.0 PL=0
MOVL C00636 V=800.0 PL=0
MOVL C00637 V=800.0 PL=0
MOVL C00638 V=800.0 PL=0
MOVL C00639 V=800.0 PL=0
MOVL C00640 V=800.0 PL=0
MOVL C00641 V=800.0 PL=0
MOVL C00642 V=800.0 PL=0
MOVL C00643 V=800.0 PL=0
MOVL C00644 V=800.0 PL=0
MOVL C00645 V=800.0 PL=0
MOVL C00646 V=800.0 PL=0
MOVL C00647 V=800.0 PL=0
MOVL C00648 V=800.0 PL=0
MOVL C00649 V=800.0 PL=0
MOVL C00650 V=800.0 PL=0
MOVL C00651 V=800.0 PL=0
MOVL C00652 V=800.0 PL=0
MOVL C00653 V=800.0 PL=0
MOVL C00654 V=800.0 PL=0
MOVL C00655 V=800.0 PL=0
MOVL C00656 V=800.0 PL=0
MOVL C00657 V=800.0 PL=0
MOVL C00658 V=800.0 PL=0
MOVL C00659 V=800.0 PL=0
MOVL C00660 V=800.0 PL=0
MOVL C00661 V=800.0 PL=0
MOVL C00662 V=800.0 PL=0
MOVL C00663 V=800.0 PL=0
MOVL C00664 V=800.0 PL=0
MOVL C00665 V=800.0 PL=0
MOVL C00666 V=800.0 PL=0
MOVL C00667 V=800.0 PL=0
MOVL C00668 V=800.0 PL=0
MOVL C00669 V=800.0 PL=0
MOVL C00670 V=800.0 PL=0
MOVL C00671 V=800.0 PL=0
MOVL C00672 V=800.0 PL=0
MOVL C00673 V=800.0 PL=0
MOVL C00674 V=800.0 PL=0
MOVL C00675 V=800.0 PL=0
MOVL C00676 V=800.0 PL=0
MOVL C00677 V=800.0 PL=0
MOVL C00678 V=800.0 PL=0
MOVL C00679 V=800.0 PL=0
MOVL C00680 V=800.0 PL=0
MOVL C00681 V=800.0 PL=0
MOVL C00682 V=800.0 PL=0
MOVL C00683 V=800.0 PL=0
MOVL C00684 V=800.0 PL=0
MOVL C00685 V=800.0 PL=0
MOVL C00686 V=800.0 PL=0
MOVL C00687 V=800.0 PL=0
MOVL C00688 V=800.0 PL=0
MOVL C00689 V=800.0 PL=0
MOVL C00690 V=800.0 PL=0
MOVL C00691 V=800.0 PL=0
MOVL C00692 V=800.0 PL=0
MOVL C00693 V=800.0 PL=0
MOVL C00694 V=800.0 PL=0
MOVL C00695 V=800.0 PL=0
MOVL C00696 V=800.0 PL=0
MOVL C00697 V=800.0 PL=0
MOVL C00698 V=800.0 PL=0
MOVL C00699 V=800.0 PL=0
MOVL C00700 V=800.0 PL=0
MOVL C00701 V=800.0 PL=0
MOVL C00702 V=800.0 PL=0
MOVL C00703 V=800.0 PL=0
MOVL C00704 V=800.0 PL=0
MOVL C00705 V=800.0 PL=0
MOVL C00706 V=800.0 PL=0
MOVL C00707 V=800.0 PL=0
MOVL C00708 V=800.0 PL=0
MOVL C00709 V=800.0 PL=0
MOVL C00710 V=800.0 PL=0
MOVL C00711 V=800.0 PL=0
MOVL C00712 V=800.0 PL=0
MOVL C00713 V=800.0 PL=0
MOVL C00714 V=800.0 PL=0
MOVL C00715 V=800.0 PL=0
MOVL C00716 V=800.0 PL=0
MOVL C00717 V=800.0 PL=0
MOVL C00718 V=800.0 PL=0
MOVL C00719 V=800.0 PL=0
MOVL C00720 V=800.0 PL=0
MOVL C00721 V=800.0 PL=0
MOVL C00722 V=800.0 PL=0
MOVL C00723 V=800.0 PL=0
MOVL C00724 V=800.0 PL=0
MOVL C00725 V=800.0 PL=0
MOVL C00726 V=800.0 PL=0
MOVL C00727 V=800.0 PL=0
MOVL C00728 V=800.0 PL=0
MOVL C00729 V=800.0 PL=0
MOVL C00730 V=800.0 PL=0
MOVL C00731 V=800.0 PL=0
MOVL C00732 V=800.0 PL=0
MOVL C00733 V=800.0 PL=0
MOVL C00734 V=800.0 PL=0
MOVL C00735 V=800.0 PL=0
MOVL C00736 V=800.0 PL=0
MOVL C00737 V=800.0 PL=0
MOVL C00738 V=800.0 PL=0
MOVL C00739 V=800.0 PL=0
MOVL C00740 V=800.0 PL=0
MOVL C00741 V=800.0 PL=0
MOVL C00742 V=800.0 PL=0
MOVL C00743 V=800.0 PL=0
MOVL C00744 V=800.0 PL=0
MOVL C00745 V=800.0 PL=0
MOVL C00746 V=800.0 PL=0
MOVL C00747 V=800.0 PL=0
MOVL C00748 V=800.0 PL=0
MOVL C00749 V=800.0 PL=0
MOVL C00750 V=800.0 PL=0
MOVL C00751 V=800.0 PL=0
MOVL C00752 V=800.0 PL=0
MOVL C00753 V=800.0 PL=0
MOVL C00754 V=800.0 PL=0
MOVL C00755 V=800.0 PL=0
MOVL C00756 V=800.0 PL=0
MOVL C00757 V=800.0 PL=0
MOVL C00758 V=800.0 PL=0
MOVL C00759 V=800.0 PL=0
MOVL C00760 V=800.0 PL=0
MOVL C00761 V=800.0 PL=0
MOVL C00762 V=800.0 PL=0
MOVL C00763 V=800.0 PL=0
MOVL C00764 V=800.0 PL=0
MOVL C00765 V=800.0 PL=0
MOVL C00766 V=800.0 PL=0
MOVL C00767 V=800.0 PL=0
MOVL C00768 V=800.0 PL=0
MOVL C00769 V=800.0 PL=0
MOVL C00770 V=800.0 PL=0
MOVL C00771 V=800.0 PL=0
MOVL C00772 V=800.0 PL=0
MOVL C00773 V=800.0 PL=0
MOVL C00774 V=800.0 PL=0
MOVL C00775 V=800.0 PL=0
MOVL C00776 V=800.0 PL=0
MOVL C00777 V=800.0 PL=0
MOVL C00778 V=800.0 PL=0
MOVL C00779 V=800.0 PL=0
MOVL C00780 V=800.0 PL=0
MOVL C00781 V=800.0 PL=0
MOVL C00782 V=800.0 PL=0
MOVL C00783 V=800.0 PL=0
MOVL C00784 V=800.0 PL=0
MOVL C00785 V=800.0 PL=0
MOVL C00786 V=800.0 PL=0
MOVL C00787 V=800.0 PL=0
MOVL C00788 V=800.0 PL=0
MOVL C00789 V=800.0 PL=0
MOVL C00790 V=800.0 PL=0
MOVL C00791 V=800.0 PL=0
MOVL C00792 V=800.0 PL=0
MOVL C00793 V=800.0 PL=0
MOVL C00794 V=800.0 PL=0
MOVL C00795 V=800.0 PL=0
MOVL C00796 V=800.0 PL=0
MOVL C00797 V=800.0 PL=0
MOVL C00798 V=800.0 PL=0
MOVL C00799 V=800.0 PL=0
MOVL C00800 V=800.0 PL=0
MOVL C00801 V=800.0 PL=0
MOVL C00802 V=800.0 PL=0
MOVL C00803 V=800.0 PL=0
MOVL C00804 V=800.0 PL=0
MOVL C00805 V=800.0 PL=0
MOVL C00806 V=800.0 PL=0
MOVL C00807 V=800.0 PL=0
MOVL C00808 V=800.0 PL=0
MOVL C00809 V=800.0 PL=0
MOVL C00810 V=800.0 PL=0
MOVL C00811 V=800.0 PL=0
MOVL C00812 V=800.0 PL=0
MOVL C00813 V=800.0 PL=0
MOVL C00814 V=800.0 PL=0
MOVL C00815 V=800.0 PL=0
MOVL C00816 V=800.0 PL=0
MOVL C00817 V=800.0 PL=0
MOVL C00818 V=800.0 PL=0
MOVL C00819 V=800.0 PL=0
MOVL C00820 V=800.0 PL=0
MOVL C00821 V=800.0 PL=0
MOVL C00822 V=800.0 PL=0
MOVL C00823 V=800.0 PL=0
MOVL C00824 V=800.0 PL=0
MOVL C00825 V=800.0 PL=0
MOVL C00826 V=800.0 PL=0
MOVL C00827 V=800.0 PL=0
MOVL C00828 V=800.0 PL=0
MOVL C00829 V=800.0 PL=0
MOVL C00830 V=800.0 PL=0
MOVL C00831 V=800.0 PL=0
MOVL C00832 V=800.0 PL=0
MOVL C00833 V=800.0 PL=0
MOVL C00834 V=800.0 PL=0
MOVL C00835 V=800.0 PL=0
MOVL C00836 V=800.0 PL=0
MOVL C00837 V=800.0 PL=0
MOVL C00838 V=800.0 PL=0
MOVL C00839 V=800.0 PL=0
MOVL C00840 V=800.0 PL=0
MOVL C00841 V=800.0 PL=0
MOVL C00842 V=800.0 PL=0
MOVL C00843 V=800.0 PL=0
MOVL C00844 V=800.0 PL=0
MOVL C00845 V=800.0 PL=0
MOVL C00846 V=800.0 PL=0
MOVL C00847 V=800.0 PL=0
MOVL C00848 V=800.0 PL=0
MOVL C00849 V=800.0 PL=0
MOVL C00850 V=800.0 PL=0
MOVL C00851 V=800.0 PL=0
MOVL C00852 V=800.0 PL=0
MOVL C00853 V=800.0 PL=0
MOVL C00854 V=800.0 PL=0
MOVL C00855 V=800.0 PL=0
MOVL C00856 V=800.0 PL=0
MOVL C00857 V=800.0 PL=0
MOVL C00858 V=800.0 PL=0
MOVL C00859 V=800.0 PL=0
MOVL C00860 V=800.0 PL=0
MOVL C00861 V=800.0 PL=0
MOVL C00862 V=800.0 PL=0
MOVL C00863 V=800.0 PL=0
MOVL C00864 V=800.0 PL=0
MOVL C00865 V=800.0 PL=0
MOVL C00866 V=800.0 PL=0
MOVL C00867 V=800.0 PL=0
MOVL C00868 V=800.0 PL=0
MOVL C00869 V=800.0 PL=0
MOVL C00870 V=800.0 PL=0
MOVL C00871 V=800.0 PL=0
MOVL C00872 V=800.0 PL=0
MOVL C00873 V=800.0 PL=0
MOVL C00874 V=800.0 PL=0
MOVL C00875 V=800.0 PL=0
MOVL C00876 V=800.0 PL=0
MOVL C00877 V=800.0 PL=0
MOVL C00878 V=800.0 PL=0
MOVL C00879 V=800.0 PL=0
MOVL C00880 V=800.0 PL=0
MOVL C00881 V=800.0 PL=0
MOVL C00882 V=800.0 PL=0
MOVL C00883 V=800.0 PL=0
MOVL C00884 V=800.0 PL=0
MOVL C00885 V=800.0 PL=0
MOVL C00886 V=800.0 PL=0
MOVL C00887 V=800.0 PL=0
MOVL C00888 V=800.0 PL=0
MOVL C00889 V=800.0 PL=0
MOVL C00890 V=800.0 PL=0
MOVL C00891 V=800.0 PL=0
MOVL C00892 V=800.0 PL=0
MOVL C00893 V=800.0 PL=0
MOVL C00894 V=800.0 PL=0
MOVL C00895 V=800.0 PL=0
MOVL C00896 V=800.0 PL=0
MOVL C00897 V=800.0 PL=0
MOVL C00898 V=800.0 PL=0
MOVL C00899 V=800.0 PL=0
MOVL C00900 V=800.0 PL=0
MOVL C00901 V=800.0 PL=0
MOVL C00902 V=800.0 PL=0
MOVL C00903 V=800.0 PL=0
MOVL C00904 V=800.0 PL=0
MOVL C00905 V=800.0 PL=0
MOVL C00906 V=800.0 PL=0
MOVL C00907 V=800.0 PL=0
MOVL C00908 V=800.0 PL=0
MOVL C00909 V=800.0 PL=0
MOVL C00910 V=800.0 PL=0
MOVL C00911 V=800.0 PL=0
MOVL C00912 V=800.0 PL=0
MOVL C00913 V=800.0 PL=0
MOVL C00914 V=800.0 PL=0
MOVL C00915 V=800.0 PL=0
MOVL C00916 V=800.0 PL=0
MOVL C00917 V=800.0 PL=0
MOVL C00918 V=800.0 PL=0
MOVL C00919 V=800.0 PL=0
MOVL C00920 V=800.0 PL=0
MOVL C00921 V=800.0 PL=0
MOVL C00922 V=800.0 PL=0
MOVL C00923 V=800.0 PL=0
MOVL C00924 V=800.0 PL=0
MOVL C00925 V=800.0 PL=0
MOVL C00926 V=800.0 PL=0
MOVL C00927 V=800.0 PL=0
MOVL C00928 V=800.0 PL=0
MOVL C00929 V=800.0 PL=0
MOVL C00930 V=800.0 PL=0
MOVL C00931 V=800.0 PL=0
MOVL C00932 V=800.0 PL=0
MOVL C00933 V=800.0 PL=0
MOVL C00934 V=800.0 PL=0
MOVL C00935 V=800.0 PL=0
MOVL C00936 V=800.0 PL=0
MOVL C00937 V=800.0 PL=0
MOVL C00938 V=800.0 PL=0
MOVL C00939 V=800.0 PL=0
MOVL C00940 V=800.0 PL=0
MOVL C00941 V=800.0 PL=0
MOVL C00942 V=800.0 PL=0
MOVL C00943 V=800.0 PL=0
MOVL C00944 V=800.0 PL=0
MOVL C00945 V=800.0 PL=0
MOVL C00946 V=800.0 PL=0
MOVL C00947 V=800.0 PL=0
MOVL C00948 V=800.0 PL=0
MOVL C00949 V=800.0 PL=0
MOVL C00950 V=800.0 PL=0
MOVL C00951 V=800.0 PL=0
MOVL C00952 V=800.0 PL=0
MOVL C00953 V=800.0 PL=0
MOVL C00954 V=800.0 PL=0
MOVL C00955 V=800.0 PL=0
MOVL C00956 V=800.0 PL=0
MOVL C00957 V=800.0 PL=0
MOVL C00958 V=800.0 PL=0
MOVL C00959 V=800.0 PL=0
MOVL C00960 V=800.0 PL=0
MOVL C00961 V=800.0 PL=0
MOVL C00962 V=800.0 PL=0
MOVL C00963 V=800.0 PL=0
MOVL C00964 V=800.0 PL=0
MOVL C00965 V=800.0 PL=0
MOVL C00966 V=800.0 PL=0
MOVL C00967 V=800.0 PL=0
MOVL C00968 V=800.0 PL=0
MOVL C00969 V=800.0 PL=0
MOVL C00970 V=800.0 PL=0
MOVL C00971 V=800.0 PL=0
MOVL C00972 V=800.0 PL=0
MOVL C00973 V=800.0 PL=0
MOVL C00974 V=800.0 PL=0
MOVL C00975 V=800.0 PL=0
MOVL C00976 V=800.0 PL=0
MOVL C00977 V=800.0 PL=0
MOVL C00978 V=800.0 PL=0
MOVL C00979 V=800.0 PL=0
MOVL C00980 V=800.0 PL=0
MOVL C00981 V=800.0 PL=0
MOVL C00982 V=800.0 PL=0
MOVL C00983 V=800.0 PL=0
MOVL C00984 V=800.0 PL=0
MOVL C00985 V=800.0 PL=0
MOVL C00986 V=800.0 PL=0
MOVL C00987 V=800.0 PL=0
MOVL C00988 V=800.0 PL=0
MOVL C00989 V=800.0 PL=0
MOVL C00990 V=800.0 PL=0
MOVL C00991 V=800.0 PL=0
MOVL C00992 V=800.0 PL=0
MOVL C00993 V=800.0 PL=0
MOVL C00994 V=800.0 PL=0
MOVL C00995 V=800.0 PL=0
MOVL C00996 V=800.0 PL=0
MOVL C00997 V=800.0 PL=0
MOVL C00998 V=800.0 PL=0
MOVL C00999 V=800.0 PL=0
MOVL C01000 V=800.0 PL=0
MOVL C01001 V=800.0 PL=0
MOVL C01002 V=800.0 PL=0
MOVL C01003 V=800.0 PL=0
MOVL C01004 V=800.0 PL=0
MOVL C01005 V=800.0 PL=0
MOVL C01006 V=800.0 PL=0
MOVL C01007 V=800.0 PL=0
MOVL C01008 V=800.0 PL=0
MOVL C01009 V=800.0 PL=0
MOVL C01010 V=800.0 PL=0
MOVL C01011 V=800.0 PL=0
MOVL C01012 V=800.0 PL=0
MOVL C01013 V=800.0 PL=0
MOVL C01014 V=800.0 PL=0
MOVL C01015 V=800.0 PL=0
MOVL C01016 V=800.0 PL=0
MOVL C01017 V=800.0 PL=0
MOVL C01018 V=800.0 PL=0
MOVL C01019 V=800.0 PL=0
MOVL C01020 V=800.0 PL=0
MOVL C01021 V=800.0 PL=0
MOVL C01022 V=800.0 PL=0
MOVL C01023 V=800.0 PL=0
MOVL C01024 V=800.0 PL=0
MOVL C01025 V=800.0 PL=0
MOVL C01026 V=800.0 PL=0
MOVL C01027 V=800.0 PL=0
MOVL C01028 V=800.0 PL=0
MOVL C01029 V=800.0 PL=0
MOVL C01030 V=800.0 PL=0
MOVL C01031 V=800.0 PL=0
MOVL C01032 V=800.0 PL=0
MOVL C01033 V=800.0 PL=0
MOVL C01034 V=800.0 PL=0
MOVL C01035 V=800.0 PL=0
MOVL C01036 V=800.0 PL=0
MOVL C01037 V=800.0 PL=0
MOVL C01038 V=800.0 PL=0
MOVL C01039 V=800.0 PL=0
MOVL C01040 V=800.0 PL=0
MOVL C01041 V=800.0 PL=0
MOVL C01042 V=800.0 PL=0
MOVL C01043 V=800.0 PL=0
MOVL C01044 V=800.0 PL=0
MOVL C01045 V=800.0 PL=0
MOVL C01046 V=800.0 PL=0
MOVL C01047 V=800.0 PL=0
MOVL C01048 V=800.0 PL=0
MOVL C01049 V=800.0 PL=0
MOVL C01050 V=800.0 PL=0
MOVL C01051 V=800.0 PL=0
MOVL C01052 V=800.0 PL=0
MOVL C01053 V=800.0 PL=0
MOVL C01054 V=800.0 PL=0
MOVL C01055 V=800.0 PL=0
MOVL C01056 V=800.0 PL=0
MOVL C01057 V=800.0 PL=0
MOVL C01058 V=800.0 PL=0
MOVL C01059 V=800.0 PL=0
MOVL C01060 V=800.0 PL=0
MOVL C01061 V=800.0 PL=0
MOVL C01062 V=800.0 PL=0
MOVL C01063 V=800.0 PL=0
MOVL C01064 V=800.0 PL=0
MOVL C01065 V=800.0 PL=0
MOVL C01066 V=800.0 PL=0
MOVL C01067 V=800.0 PL=0
MOVL C01068 V=800.0 PL=0
MOVL C01069 V=800.0 PL=0
MOVL C01070 V=800.0 PL=0
MOVL C01071 V=800.0 PL=0
MOVL C01072 V=800.0 PL=0
MOVL C01073 V=800.0 PL=0
MOVL C01074 V=800.0 PL=0
MOVL C01075 V=800.0 PL=0
MOVL C01076 V=800.0 PL=0
MOVL C01077 V=800.0 PL=0
MOVL C01078 V=800.0 PL=0
MOVL C01079 V=800.0 PL=0
MOVL C01080 V=800.0 PL=0
MOVL C01081 V=800.0 PL=0
MOVL C01082 V=800.0 PL=0
MOVL C01083 V=800.0 PL=0
MOVL C01084 V=800.0 PL=0
MOVL C01085 V=800.0 PL=0
MOVL C01086 V=800.0 PL=0
MOVL C01087 V=800.0 PL=0
MOVL C01088 V=800.0 PL=0
MOVL C01089 V=800.0 PL=0
MOVL C01090 V=800.0 PL=0
MOVL C01091 V=800.0 PL=0
MOVL C01092 V=800.0 PL=0
MOVL C01093 V=800.0 PL=0
MOVL C01094 V=800.0 PL=0
MOVL C01095 V=800.0 PL=0
MOVL C01096 V=800.0 PL=0
MOVL C01097 V=800.0 PL=0
MOVL C01098 V=800.0 PL=0
MOVL C01099 V=800.0 PL=0
MOVL C01100 V=800.0 PL=0
MOVL C01101 V=800.0 PL=0
MOVL C01102 V=800.0 PL=0
MOVL C01103 V=800.0 PL=0
MOVL C01104 V=800.0 PL=0
MOVL C01105 V=800.0 PL=0
MOVL C01106 V=800.0 PL=0
MOVL C01107 V=800.0 PL=0
MOVL C01108 V=800.0 PL=0
MOVL C01109 V=800.0 PL=0
MOVL C01110 V=800.0 PL=0
MOVL C01111 V=800.0 PL=0
MOVL C01112 V=800.0 PL=0
MOVL C01113 V=800.0 PL=0
MOVL C01114 V=800.0 PL=0
MOVL C01115 V=800.0 PL=0
MOVL C01116 V=800.0 PL=0
MOVL C01117 V=800.0 PL=0
MOVL C01118 V=800.0 PL=0
MOVL C01119 V=800.0 PL=0
MOVL C01120 V=800.0 PL=0
MOVL C01121 V=800.0 PL=0
MOVL C01122 V=800.0 PL=0
MOVL C01123 V=800.0 PL=0
MOVL C01124 V=800.0 PL=0
MOVL C01125 V=800.0 PL=0
MOVL C01126 V=800.0 PL=0
MOVL C01127 V=800.0 PL=0
MOVL C01128 V=800.0 PL=0
MOVL C01129 V=800.0 PL=0
MOVL C01130 V=800.0 PL=0
MOVL C01131 V=800.0 PL=0
MOVL C01132 V=800.0 PL=0
MOVL C01133 V=800.0 PL=0
MOVL C01134 V=800.0 PL=0
MOVL C01135 V=800.0 PL=0
MOVL C01136 V=800.0 PL=0
MOVL C01137 V=800.0 PL=0
MOVL C01138 V=800.0 PL=0
MOVL C01139 V=800.0 PL=0
MOVL C01140 V=800.0 PL=0
MOVL C01141 V=800.0 PL=0
MOVL C01142 V=800.0 PL=0
MOVL C01143 V=800.0 PL=0
MOVL C01144 V=800.0 PL=0
MOVL C01145 V=800.0 PL=0
MOVL C01146 V=800.0 PL=0
MOVL C01147 V=800.0 PL=0
MOVL C01148 V=800.0 PL=0
MOVL C01149 V=800.0 PL=0
MOVL C01150 V=800.0 PL=0
MOVL C01151 V=800.0 PL=0
MOVL C01152 V=800.0 PL=0
MOVL C01153 V=800.0 PL=0
MOVL C01154 V=800.0 PL=0
MOVL C01155 V=800.0 PL=0
MOVL C01156 V=800.0 PL=0
MOVL C01157 V=800.0 PL=0
MOVL C01158 V=800.0 PL=0
MOVL C01159 V=800.0 PL=0
MOVL C01160 V=800.0 PL=0
MOVL C01161 V=800.0 PL=0
MOVL C01162 V=800.0 PL=0
MOVL C01163 V=800.0 PL=0
MOVL C01164 V=800.0 PL=0
MOVL C01165 V=800.0 PL=0
MOVL C01166 V=800.0 PL=0
MOVL C01167 V=800.0 PL=0
MOVL C01168 V=800.0 PL=0
MOVL C01169 V=800.0 PL=0
MOVL C01170 V=800.0 PL=0
MOVL C01171 V=800.0 PL=0
MOVL C01172 V=800.0 PL=0
MOVL C01173 V=800.0 PL=0
MOVL C01174 V=800.0 PL=0
MOVL C01175 V=800.0 PL=0
MOVL C01176 V=800.0 PL=0
MOVL C01177 V=800.0 PL=0
MOVL C01178 V=800.0 PL=0
MOVL C01179 V=800.0 PL=0
MOVL C01180 V=800.0 PL=0
MOVL C01181 V=800.0 PL=0
MOVL C01182 V=800.0 PL=0
MOVL C01183 V=800.0 PL=0
MOVL C01184 V=800.0 PL=0
MOVL C01185 V=800.0 PL=0
MOVL C01186 V=800.0 PL=0
MOVL C01187 V=800.0 PL=0
MOVL C01188 V=800.0 PL=0
MOVL C01189 V=800.0 PL=0
MOVL C01190 V=800.0 PL=0
MOVL C01191 V=800.0 PL=0
MOVL C01192 V=800.0 PL=0
MOVL C01193 V=800.0 PL=0
MOVL C01194 V=800.0 PL=0
MOVL C01195 V=800.0 PL=0
MOVL C01196 V=800.0 PL=0
MOVL C01197 V=800.0 PL=0
MOVL C01198 V=800.0 PL=0
MOVL C01199 V=800.0 PL=0
MOVL C01200 V=800.0 PL=0
MOVL C01201 V=800.0 PL=0
MOVL C01202 V=800.0 PL=0
MOVL C01203 V=800.0 PL=0
MOVL C01204 V=800.0 PL=0
MOVL C01205 V=800.0 PL=0
MOVL C01206 V=800.0 PL=0
MOVL C01207 V=800.0 PL=0
MOVL C01208 V=800.0 PL=0
MOVL C01209 V=800.0 PL=0
MOVL C01210 V=800.0 PL=0
MOVL C01211 V=800.0 PL=0
MOVL C01212 V=800.0 PL=0
MOVL C01213 V=800.0 PL=0
MOVL C01214 V=800.0 PL=0
MOVL C01215 V=800.0 PL=0
MOVL C01216 V=800.0 PL=0
MOVL C01217 V=800.0 PL=0
MOVL C01218 V=800.0 PL=0
MOVL C01219 V=800.0 PL=0
MOVL C01220 V=800.0 PL=0
MOVL C01221 V=800.0 PL=0
MOVL C01222 V=800.0 PL=0
MOVL C01223 V=800.0 PL=0
MOVL C01224 V=800.0 PL=0
MOVL C01225 V=800.0 PL=0
MOVL C01226 V=800.0 PL=0
MOVL C01227 V=800.0 PL=0
MOVL C01228 V=800.0 PL=0
MOVL C01229 V=800.0 PL=0
MOVL C01230 V=800.0 PL=0
MOVL C01231 V=800.0 PL=0
MOVL C01232 V=800.0 PL=0
MOVL C01233 V=800.0 PL=0
MOVL C01234 V=800.0 PL=0
MOVL C01235 V=800.0 PL=0
MOVL C01236 V=800.0 PL=0
MOVL C01237 V=800.0 PL=0
MOVL C01238 V=800.0 PL=0
MOVL C01239 V=800.0 PL=0
MOVL C01240 V=800.0 PL=0
MOVL C01241 V=800.0 PL=0
MOVL C01242 V=800.0 PL=0
MOVL C01243 V=800.0 PL=0
MOVL C01244 V=800.0 PL=0
MOVL C01245 V=800.0 PL=0
MOVL C01246 V=800.0 PL=0
MOVL C01247 V=800.0 PL=0
MOVL C01248 V=800.0 PL=0
MOVL C01249 V=800.0 PL=0
MOVL C01250 V=800.0 PL=0
MOVL C01251 V=800.0 PL=0
MOVL C01252 V=800.0 PL=0
MOVL C01253 V=800.0 PL=0
MOVL C01254 V=800.0 PL=0
MOVL C01255 V=800.0 PL=0
MOVL C01256 V=800.0 PL=0
MOVL C01257 V=800.0 PL=0
MOVL C01258 V=800.0 PL=0
MOVL C01259 V=800.0 PL=0
MOVL C01260 V=800.0 PL=0
MOVL C01261 V=800.0 PL=0
MOVL C01262 V=800.0 PL=0
MOVL C01263 V=800.0 PL=0
MOVL C01264 V=800.0 PL=0
MOVL C01265 V=800.0 PL=0
MOVL C01266 V=800.0 PL=0
MOVL C01267 V=800.0 PL=0
MOVL C01268 V=800.0 PL=0
MOVL C01269 V=800.0 PL=0
MOVL C01270 V=800.0 PL=0
MOVL C01271 V=800.0 PL=0
MOVL C01272 V=800.0 PL=0
MOVL C01273 V=800.0 PL=0
MOVL C01274 V=800.0 PL=0
MOVL C01275 V=800.0 PL=0
MOVL C01276 V=800.0 PL=0
MOVL C01277 V=800.0 PL=0
MOVL C01278 V=800.0 PL=0
MOVL C01279 V=800.0 PL=0
MOVL C01280 V=800.0 PL=0
MOVL C01281 V=800.0 PL=0
MOVL C01282 V=800.0 PL=0
MOVL C01283 V=800.0 PL=0
MOVL C01284 V=800.0 PL=0
MOVL C01285 V=800.0 PL=0
MOVL C01286 V=800.0 PL=0
MOVL C01287 V=800.0 PL=0
MOVL C01288 V=800.0 PL=0
MOVL C01289 V=800.0 PL=0
MOVL C01290 V=800.0 PL=0
MOVL C01291 V=800.0 PL=0
MOVL C01292 V=800.0 PL=0
MOVL C01293 V=800.0 PL=0
MOVL C01294 V=800.0 PL=0
MOVL C01295 V=800.0 PL=0
MOVL C01296 V=800.0 PL=0
MOVL C01297 V=800.0 PL=0
MOVL C01298 V=800.0 PL=0
MOVL C01299 V=800.0 PL=0
MOVL C01300 V=800.0 PL=0
MOVL C01301 V=800.0 PL=0
MOVL C01302 V=800.0 PL=0
MOVL C01303 V=800.0 PL=0
MOVL C01304 V=800.0 PL=0
MOVL C01305 V=800.0 PL=0
MOVL C01306 V=800.0 PL=0
MOVL C01307 V=800.0 PL=0
MOVL C01308 V=800.0 PL=0
MOVL C01309 V=800.0 PL=0
MOVL C01310 V=800.0 PL=0
MOVL C01311 V=800.0 PL=0
MOVL C01312 V=800.0 PL=0
MOVL C01313 V=800.0 PL=0
MOVL C01314 V=800.0 PL=0
MOVL C01315 V=800.0 PL=0
MOVL C01316 V=800.0 PL=0
MOVL C01317 V=800.0 PL=0
MOVL C01318 V=800.0 PL=0
MOVL C01319 V=800.0 PL=0
MOVL C01320 V=800.0 PL=0
MOVL C01321 V=800.0 PL=0
MOVL C01322 V=800.0 PL=0
MOVL C01323 V=800.0 PL=0
MOVL C01324 V=800.0 PL=0
MOVL C01325 V=800.0 PL=0
MOVL C01326 V=800.0 PL=0
MOVL C01327 V=800.0 PL=0
MOVL C01328 V=800.0 PL=0
MOVL C01329 V=800.0 PL=0
MOVL C01330 V=800.0 PL=0
MOVL C01331 V=800.0 PL=0
MOVL C01332 V=800.0 PL=0
MOVL C01333 V=800.0 PL=0
MOVL C01334 V=800.0 PL=0
MOVL C01335 V=800.0 PL=0
MOVL C01336 V=800.0 PL=0
MOVL C01337 V=800.0 PL=0
MOVL C01338 V=800.0 PL=0
MOVL C01339 V=800.0 PL=0
MOVL C01340 V=800.0 PL=0
MOVL C01341 V=800.0 PL=0
MOVL C01342 V=800.0 PL=0
MOVL C01343 V=800.0 PL=0
MOVL C01344 V=800.0 PL=0
MOVL C01345 V=800.0 PL=0
MOVL C01346 V=800.0 PL=0
MOVL C01347 V=800.0 PL=0
MOVL C01348 V=800.0 PL=0
MOVL C01349 V=800.0 PL=0
MOVL C01350 V=800.0 PL=0
MOVL C01351 V=800.0 PL=0
MOVL C01352 V=800.0 PL=0
MOVL C01353 V=800.0 PL=0
MOVL C01354 V=800.0 PL=0
MOVL C01355 V=800.0 PL=0
MOVL C01356 V=800.0 PL=0
MOVL C01357 V=800.0 PL=0
MOVL C01358 V=800.0 PL=0
MOVL C01359 V=800.0 PL=0
MOVL C01360 V=800.0 PL=0
MOVL C01361 V=800.0 PL=0
MOVL C01362 V=800.0 PL=0
MOVL C01363 V=800.0 PL=0
MOVL C01364 V=800.0 PL=0
MOVL C01365 V=800.0 PL=0
MOVL C01366 V=800.0 PL=0
MOVL C01367 V=800.0 PL=0
MOVL C01368 V=800.0 PL=0
MOVL C01369 V=800.0 PL=0
MOVL C01370 V=800.0 PL=0
MOVL C01371 V=800.0 PL=0
MOVL C01372 V=800.0 PL=0
MOVL C01373 V=800.0 PL=0
MOVL C01374 V=800.0 PL=0
MOVL C01375 V=800.0 PL=0
MOVL C01376 V=800.0 PL=0
MOVL C01377 V=800.0 PL=0
MOVL C01378 V=800.0 PL=0
MOVL C01379 V=800.0 PL=0
MOVL C01380 V=800.0 PL=0
MOVL C01381 V=800.0 PL=0
MOVL C01382 V=800.0 PL=0
MOVL C01383 V=800.0 PL=0
MOVL C01384 V=800.0 PL=0
MOVL C01385 V=800.0 PL=0
MOVL C01386 V=800.0 PL=0
MOVL C01387 V=800.0 PL=0
MOVL C01388 V=800.0 PL=0
MOVL C01389 V=800.0 PL=0
MOVL C01390 V=800.0 PL=0
MOVL C01391 V=800.0 PL=0
MOVL C01392 V=800.0 PL=0
MOVL C01393 V=800.0 PL=0
MOVL C01394 V=800.0 PL=0
MOVL C01395 V=800.0 PL=0
MOVL C01396 V=800.0 PL=0
MOVL C01397 V=800.0 PL=0
MOVL C01398 V=800.0 PL=0
MOVL C01399 V=800.0 PL=0
MOVL C01400 V=800.0 PL=0
MOVL C01401 V=800.0 PL=0
MOVL C01402 V=800.0 PL=0
MOVL C01403 V=800.0 PL=0
MOVL C01404 V=800.0 PL=0
MOVL C01405 V=800.0 PL=0
MOVL C01406 V=800.0 PL=0
MOVL C01407 V=800.0 PL=0
MOVL C01408 V=800.0 PL=0
MOVL C01409 V=800.0 PL=0
MOVL C01410 V=800.0 PL=0
MOVL C01411 V=800.0 PL=0
MOVL C01412 V=800.0 PL=0
MOVL C01413 V=800.0 PL=0
MOVL C01414 V=800.0 PL=0
MOVL C01415 V=800.0 PL=0
MOVL C01416 V=800.0 PL=0
MOVL C01417 V=800.0 PL=0
MOVL C01418 V=800.0 PL=0
MOVL C01419 V=800.0 PL=0
MOVL C01420 V=800.0 PL=0
MOVL C01421 V=800.0 PL=0
MOVL C01422 V=800.0 PL=0
MOVL C01423 V=800.0 PL=0
MOVL C01424 V=800.0 PL=0
MOVL C01425 V=800.0 PL=0
MOVL C01426 V=800.0 PL=0
MOVL C01427 V=800.0 PL=0
MOVL C01428 V=800.0 PL=0
MOVL C01429 V=800.0 PL=0
MOVL C01430 V=800.0 PL=0
MOVL C01431 V=800.0 PL=0
MOVL C01432 V=800.0 PL=0
MOVL C01433 V=800.0 PL=0
MOVL C01434 V=800.0 PL=0
MOVL C01435 V=800.0 PL=0
MOVL C01436 V=800.0 PL=0
MOVL C01437 V=800.0 PL=0
MOVL C01438 V=800.0 PL=0
MOVL C01439 V=800.0 PL=0
MOVL C01440 V=800.0 PL=0
MOVL C01441 V=800.0 PL=0
MOVL C01442 V=800.0 PL=0
MOVL C01443 V=800.0 PL=0
MOVL C01444 V=800.0 PL=0
MOVL C01445 V=800.0 PL=0
MOVL C01446 V=800.0 PL=0
MOVL C01447 V=800.0 PL=0
MOVL C01448 V=800.0 PL=0
MOVL C01449 V=800.0 PL=0
MOVL C01450 V=800.0 PL=0
MOVL C01451 V=800.0 PL=0
MOVL C01452 V=800.0 PL=0
MOVL C01453 V=800.0 PL=0
MOVL C01454 V=800.0 PL=0
MOVL C01455 V=800.0 PL=0
MOVL C01456 V=800.0 PL=0
MOVL C01457 V=800.0 PL=0
MOVL C01458 V=800.0 PL=0
MOVL C01459 V=800.0 PL=0
MOVL C01460 V=800.0 PL=0
MOVL C01461 V=800.0 PL=0
MOVL C01462 V=800.0 PL=0
MOVL C01463 V=800.0 PL=0
MOVL C01464 V=800.0 PL=0
MOVL C01465 V=800.0 PL=0
MOVL C01466 V=800.0 PL=0
MOVL C01467 V=800.0 PL=0
MOVL C01468 V=800.0 PL=0
MOVL C01469 V=800.0 PL=0
MOVL C01470 V=800.0 PL=0
MOVL C01471 V=800.0 PL=0
MOVL C01472 V=800.0 PL=0
MOVL C01473 V=800.0 PL=0
MOVL C01474 V=800.0 PL=0
MOVL C01475 V=800.0 PL=0
MOVL C01476 V=800.0 PL=0
MOVL C01477 V=800.0 PL=0
MOVL C01478 V=800.0 PL=0
MOVL C01479 V=800.0 PL=0
MOVL C01480 V=800.0 PL=0
MOVL C01481 V=800.0 PL=0
MOVL C01482 V=800.0 PL=0
MOVL C01483 V=800.0 PL=0
MOVL C01484 V=800.0 PL=0
MOVL C01485 V=800.0 PL=0
MOVL C01486 V=800.0 PL=0
MOVL C01487 V=800.0 PL=0
MOVL C01488 V=800.0 PL=0
MOVL C01489 V=800.0 PL=0
MOVL C01490 V=800.0 PL=0
MOVL C01491 V=800.0 PL=0
MOVL C01492 V=800.0 PL=0
MOVL C01493 V=800.0 PL=0
MOVL C01494 V=800.0 PL=0
MOVL C01495 V=800.0 PL=0
MOVL C01496 V=800.0 PL=0
MOVL C01497 V=800.0 PL=0
MOVL C01498 V=800.0 PL=0
MOVL C01499 V=800.0 PL=0
MOVL C01500 V=800.0 PL=0
MOVL C01501 V=800.0 PL=0
MOVL C01502 V=800.0 PL=0
MOVL C01503 V=800.0 PL=0
MOVL C01504 V=800.0 PL=0
MOVL C01505 V=800.0 PL=0
MOVL C01506 V=800.0 PL=0
MOVL C01507 V=800.0 PL=0
MOVL C01508 V=800.0 PL=0
MOVL C01509 V=800.0 PL=0
MOVL C01510 V=800.0 PL=0
MOVL C01511 V=800.0 PL=0
MOVL C01512 V=800.0 PL=0
MOVL C01513 V=800.0 PL=0
MOVL C01514 V=800.0 PL=0
MOVL C01515 V=800.0 PL=0
MOVL C01516 V=800.0 PL=0
MOVL C01517 V=800.0 PL=0
MOVL C01518 V=800.0 PL=0
MOVL C01519 V=800.0 PL=0
MOVL C01520 V=800.0 PL=0
MOVL C01521 V=800.0 PL=0
MOVL C01522 V=800.0 PL=0
MOVL C01523 V=800.0 PL=0
MOVL C01524 V=800.0 PL=0
MOVL C01525 V=800.0 PL=0
MOVL C01526 V=800.0 PL=0
MOVL C01527 V=800.0 PL=0
MOVL C01528 V=800.0 PL=0
MOVL C01529 V=800.0 PL=0
MOVL C01530 V=800.0 PL=0
MOVL C01531 V=800.0 PL=0
MOVL C01532 V=800.0 PL=0
MOVL C01533 V=800.0 PL=0
MOVL C01534 V=800.0 PL=0
MOVL C01535 V=800.0 PL=0
MOVL C01536 V=800.0 PL=0
MOVL C01537 V=800.0 PL=0
MOVL C01538 V=800.0 PL=0
MOVL C01539 V=800.0 PL=0
MOVL C01540 V=800.0 PL=0
MOVL C01541 V=800.0 PL=0
MOVL C01542 V=800.0 PL=0
MOVL C01543 V=800.0 PL=0
MOVL C01544 V=800.0 PL=0
MOVL C01545 V=800.0 PL=0
MOVL C01546 V=800.0 PL=0
MOVL C01547 V=800.0 PL=0
MOVL C01548 V=800.0 PL=0
MOVL C01549 V=800.0 PL=0
MOVL C01550 V=800.0 PL=0
MOVL C01551 V=800.0 PL=0
MOVL C01552 V=800.0 PL=0
MOVL C01553 V=800.0 PL=0
MOVL C01554 V=800.0 PL=0
MOVL C01555 V=800.0 PL=0
MOVL C01556 V=800.0 PL=0
MOVL C01557 V=800.0 PL=0
MOVL C01558 V=800.0 PL=0
MOVL C01559 V=800.0 PL=0
MOVL C01560 V=800.0 PL=0
MOVL C01561 V=800.0 PL=0
MOVL C01562 V=800.0 PL=0
MOVL C01563 V=800.0 PL=0
MOVL C01564 V=800.0 PL=0
MOVL C01565 V=800.0 PL=0
MOVL C01566 V=800.0 PL=0
MOVL C01567 V=800.0 PL=0
MOVL C01568 V=800.0 PL=0
MOVL C01569 V=800.0 PL=0
MOVL C01570 V=800.0 PL=0
MOVL C01571 V=800.0 PL=0
MOVL C01572 V=800.0 PL=0
MOVL C01573 V=800.0 PL=0
MOVL C01574 V=800.0 PL=0
MOVL C01575 V=800.0 PL=0
MOVL C01576 V=800.0 PL=0
MOVL C01577 V=800.0 PL=0
MOVL C01578 V=800.0 PL=0
MOVL C01579 V=800.0 PL=0
MOVL C01580 V=800.0 PL=0
MOVL C01581 V=800.0 PL=0
MOVL C01582 V=800.0 PL=0
MOVL C01583 V=800.0 PL=0
MOVL C01584 V=800.0 PL=0
MOVL C01585 V=800.0 PL=0
MOVL C01586 V=800.0 PL=0
MOVL C01587 V=800.0 PL=0
MOVL C01588 V=800.0 PL=0
MOVL C01589 V=800.0 PL=0
MOVL C01590 V=800.0 PL=0
MOVL C01591 V=800.0 PL=0
MOVL C01592 V=800.0 PL=0
MOVL C01593 V=800.0 PL=0
MOVL C01594 V=800.0 PL=0
MOVL C01595 V=800.0 PL=0
MOVL C01596 V=800.0 PL=0
MOVL C01597 V=800.0 PL=0
MOVL C01598 V=800.0 PL=0
MOVL C01599 V=800.0 PL=0
MOVL C01600 V=800.0 PL=0
MOVL C01601 V=800.0 PL=0
MOVL C01602 V=800.0 PL=0
MOVL C01603 V=800.0 PL=0
MOVL C01604 V=800.0 PL=0
MOVL C01605 V=800.0 PL=0
MOVL C01606 V=800.0 PL=0
MOVL C01607 V=800.0 PL=0
MOVL C01608 V=800.0 PL=0
MOVL C01609 V=800.0 PL=0
MOVL C01610 V=800.0 PL=0
MOVL C01611 V=800.0 PL=0
MOVL C01612 V=800.0 PL=0
MOVL C01613 V=800.0 PL=0
MOVL C01614 V=800.0 PL=0
MOVL C01615 V=800.0 PL=0
MOVL C01616 V=800.0 PL=0
MOVL C01617 V=800.0 PL=0
MOVL C01618 V=800.0 PL=0
MOVL C01619 V=800.0 PL=0
MOVL C01620 V=800.0 PL=0
MOVL C01621 V=800.0 PL=0
MOVL C01622 V=800.0 PL=0
MOVL C01623 V=800.0 PL=0
MOVL C01624 V=800.0 PL=0
MOVL C01625 V=800.0 PL=0
MOVL C01626 V=800.0 PL=0
MOVL C01627 V=800.0 PL=0
MOVL C01628 V=800.0 PL=0
MOVL C01629 V=800.0 PL=0
MOVL C01630 V=800.0 PL=0
MOVL C01631 V=800.0 PL=0
MOVL C01632 V=800.0 PL=0
MOVL C01633 V=800.0 PL=0
MOVL C01634 V=800.0 PL=0
MOVL C01635 V=800.0 PL=0
MOVL C01636 V=800.0 PL=0
MOVL C01637 V=800.0 PL=0
MOVL C01638 V=800.0 PL=0
MOVL C01639 V=800.0 PL=0
MOVL C01640 V=800.0 PL=0
MOVL C01641 V=800.0 PL=0
MOVL C01642 V=800.0 PL=0
MOVL C01643 V=800.0 PL=0
MOVL C01644 V=800.0 PL=0
MOVL C01645 V=800.0 PL=0
MOVL C01646 V=800.0 PL=0
MOVL C01647 V=800.0 PL=0
MOVL C01648 V=800.0 PL=0
MOVL C01649 V=800.0 PL=0
MOVL C01650 V=800.0 PL=0
MOVL C01651 V=800.0 PL=0
MOVL C01652 V=800.0 PL=0
MOVL C01653 V=800.0 PL=0
MOVL C01654 V=800.0 PL=0
MOVL C01655 V=800.0 PL=0
MOVL C01656 V=800.0 PL=0
MOVL C01657 V=800.0 PL=0
MOVL C01658 V=800.0 PL=0
MOVL C01659 V=800.0 PL=0
MOVL C01660 V=800.0 PL=0
MOVL C01661 V=800.0 PL=0
MOVL C01662 V=800.0 PL=0
MOVL C01663 V=800.0 PL=0
MOVL C01664 V=800.0 PL=0
MOVL C01665 V=800.0 PL=0
MOVL C01666 V=800.0 PL=0
MOVL C01667 V=800.0 PL=0
MOVL C01668 V=800.0 PL=0
MOVL C01669 V=800.0 PL=0
MOVL C01670 V=800.0 PL=0
MOVL C01671 V=800.0 PL=0
MOVL C01672 V=800.0 PL=0
MOVL C01673 V=800.0 PL=0
MOVL C01674 V=800.0 PL=0
MOVL C01675 V=800.0 PL=0
MOVL C01676 V=800.0 PL=0
MOVL C01677 V=800.0 PL=0
MOVL C01678 V=800.0 PL=0
MOVL C01679 V=800.0 PL=0
MOVL C01680 V=800.0 PL=0
MOVL C01681 V=800.0 PL=0
MOVL C01682 V=800.0 PL=0
MOVL C01683 V=800.0 PL=0
MOVL C01684 V=800.0 PL=0
MOVL C01685 V=800.0 PL=0
MOVL C01686 V=800.0 PL=0
MOVL C01687 V=800.0 PL=0
MOVL C01688 V=800.0 PL=0
MOVL C01689 V=800.0 PL=0
MOVL C01690 V=800.0 PL=0
MOVL C01691 V=800.0 PL=0
MOVL C01692 V=800.0 PL=0
MOVL C01693 V=800.0 PL=0
MOVL C01694 V=800.0 PL=0
MOVL C01695 V=800.0 PL=0
MOVL C01696 V=800.0 PL=0
MOVL C01697 V=800.0 PL=0
MOVL C01698 V=800.0 PL=0
MOVL C01699 V=800.0 PL=0
MOVL C01700 V=800.0 PL=0
MOVL C01701 V=800.0 PL=0
MOVL C01702 V=800.0 PL=0
MOVL C01703 V=800.0 PL=0
MOVL C01704 V=800.0 PL=0
MOVL C01705 V=800.0 PL=0
MOVL C01706 V=800.0 PL=0
MOVL C01707 V=800.0 PL=0
MOVL C01708 V=800.0 PL=0
MOVL C01709 V=800.0 PL=0
MOVL C01710 V=800.0 PL=0
MOVL C01711 V=800.0 PL=0
MOVL C01712 V=800.0 PL=0
MOVL C01713 V=800.0 PL=0
MOVL C01714 V=800.0 PL=0
MOVL C01715 V=800.0 PL=0
MOVL C01716 V=800.0 PL=0
MOVL C01717 V=800.0 PL=0
MOVL C01718 V=800.0 PL=0
MOVL C01719 V=800.0 PL=0
MOVL C01720 V=800.0 PL=0
MOVL C01721 V=800.0 PL=0
MOVL C01722 V=800.0 PL=0
MOVL C01723 V=800.0 PL=0
MOVL C01724 V=800.0 PL=0
MOVL C01725 V=800.0 PL=0
MOVL C01726 V=800.0 PL=0
MOVL C01727 V=800.0 PL=0
MOVL C01728 V=800.0 PL=0
MOVL C01729 V=800.0 PL=0
MOVL C01730 V=800.0 PL=0
MOVL C01731 V=800.0 PL=0
MOVL C01732 V=800.0 PL=0
MOVL C01733 V=800.0 PL=0
MOVL C01734 V=800.0 PL=0
MOVL C01735 V=800.0 PL=0
MOVL C01736 V=800.0 PL=0
MOVL C01737 V=800.0 PL=0
MOVL C01738 V=800.0 PL=0
MOVL C01739 V=800.0 PL=0
MOVL C01740 V=800.0 PL=0
MOVL C01741 V=800.0 PL=0
MOVL C01742 V=800.0 PL=0
MOVL C01743 V=800.0 PL=0
MOVL C01744 V=800.0 PL=0
MOVL C01745 V=800.0 PL=0
MOVL C01746 V=800.0 PL=0
MOVL C01747 V=800.0 PL=0
MOVL C01748 V=800.0 PL=0
MOVL C01749 V=800.0 PL=0
MOVL C01750 V=800.0 PL=0
MOVL C01751 V=800.0 PL=0
MOVL C01752 V=800.0 PL=0
MOVL C01753 V=800.0 PL=0
MOVL C01754 V=800.0 PL=0
MOVL C01755 V=800.0 PL=0
MOVL C01756 V=800.0 PL=0
MOVL C01757 V=800.0 PL=0
MOVL C01758 V=800.0 PL=0
MOVL C01759 V=800.0 PL=0
MOVL C01760 V=800.0 PL=0
MOVL C01761 V=800.0 PL=0
